IF (NOT(gSystemPrimary.OperatingMode.Stopped)) THEN
	//gMessageManager.register(lCode:=cMCAdviseFunctionalModeNotStationary);
	lDiagnostic := cFunctionalDiagnosticNotStationary;
	request := lDiagnostic;
	RETURN;
END_IF

IF (NOT(lMode.leave())) THEN
	//gMessageManager.register(lCode:=cMCAdviseFunctionalModeWaitingOnPreviousToExit);
	lDiagnostic := cFunctionalDiagnosticWaitingOnPreviousToExit;
	request := lDiagnostic;
	RETURN;
END_IF

lMode REF= mode;
lRequested := TRUE;

IF (NOT(lMode.enter())) THEN
	//gMessageManager.register(lCode:=cMCAdviseFunctionalModeNotYetActive);
	lDiagnostic := cFunctionalDiagnosticNotYetActive;
	request := lDiagnostic;
	RETURN;
END_IF

lDiagnostic := cFunctionalDiagnosticOK;
request := lDiagnostic;


                
END_METHOD

PROPERTY Active : BOOL
GET
                    Active := Mode.Active;
                  
END_GET
END_PROPERTY

(* {attribute 'monitoring' := 'call'} *)
PROPERTY CurrentMode : t_functional_mode
GET
                    CurrentMode := lMode.Mode;


                  
END_GET
SET
                    request(CurrentMode);
                  
END_SET
END_PROPERTY

(* {attribute 'monitoring' := 'call'} *)
PROPERTY Diagnostic : t_functional_diagnostic
GET
                    Diagnostic := lDiagnostic;
                  
END_GET
END_PROPERTY

PROPERTY Mode : REFERENCE TO FunctionalMode
GET
                    Mode REF= lMode;

                  
END_GET
END_PROPERTY

PROPERTY Requested : BOOL
GET
                    Requested := lRequested;
                  
END_GET
END_PROPERTY

PROPERTY TypeToken : t_medium_string
GET
                    TypeToken := 'FuncModeCntrl';
                  
END_GET
END_PROPERTY
END_FUNCTION_BLOCK

FUNCTION_BLOCK FunctionalModeDefault EXTENDS FunctionalMode

            ;
          

METHOD initialize
                  SUPER^.initialize();

lMode := cFunctionalModeDefault;

                
END_METHOD
END_FUNCTION_BLOCK

FUNCTION_BLOCK FunctionalModeLift EXTENDS FunctionalMode

            ;
          

METHOD initialize
                  SUPER^.initialize();

lMode := cFunctionalModeLift;

                
END_METHOD
END_FUNCTION_BLOCK

FUNCTION_BLOCK FunctionalModeTravel EXTENDS FunctionalMode

            ;
          

METHOD initialize
                  SUPER^.initialize();

lMode := cFunctionalModeTravel;

                
END_METHOD
END_FUNCTION_BLOCK

FUNCTION_BLOCK SteerAPositionInterlock EXTENDS WrapperScaledInterlock
  VAR CONSTANT
    cOuterRegion : t_percentage := 1.0;
    cInnerRegion : t_percentage := 0.98;
    cInnerValue : t_percentage := 1.0;
    cOuterValue : t_percentage := 0.0;
    cZeroThreshold : t_percentage := 0.03;
  END_VAR

            ;
          

METHOD initialize
                  Name := 'iSteerAPos';

Input REF= gSystemPrimary.CANOpenMasterDrivePrimary.SteerAngleA.PositionObject;

lTransform.InnerRegion := cInnerRegion;
lTransform.OuterRegion := cOuterRegion;
lTransform.InnerValue := cInnerValue;
lTransform.OuterValue := cOuterValue;

Client.registerServer(gSystemPrimary.Steering.WheelA.Interlock);
Client.ScalingContext REF= gSystemPrimary.Steering.WheelA.InputObject;
Client.ZeroThreshold := cZeroThreshold;
Sign := -1.0;

SUPER^.initialize();

                
END_METHOD
END_FUNCTION_BLOCK

FUNCTION_BLOCK SteerBPositionInterlock EXTENDS WrapperScaledInterlock
  VAR CONSTANT
    cOuterRegion : t_percentage := 1.0;
    cInnerRegion : t_percentage := 0.98;
    cInnerValue : t_percentage := 1.0;
    cOuterValue : t_percentage := 0.0;
    cZeroThreshold : t_percentage := 0.03;
  END_VAR

            ;
          

METHOD initialize
                  Name := 'iSteerBPos';

Input REF= gSystemPrimary.CANOpenMasterDrivePrimary.SteerAngleB.PositionObject;

lTransform.InnerRegion := cInnerRegion;
lTransform.OuterRegion := cOuterRegion;
lTransform.InnerValue := cInnerValue;
lTransform.OuterValue := cOuterValue;

Client.registerServer(gSystemPrimary.Steering.WheelB.Interlock);
Client.ScalingContext REF= gSystemPrimary.Steering.WheelB.InputObject;
Client.ZeroThreshold := cZeroThreshold;
Sign := -1.0;

SUPER^.initialize();

                
END_METHOD
END_FUNCTION_BLOCK

FUNCTION_BLOCK SteerCPositionInterlock EXTENDS WrapperScaledInterlock
  VAR CONSTANT
    cOuterRegion : t_percentage := 1.0;
    cInnerRegion : t_percentage := 0.98;
    cInnerValue : t_percentage := 1.0;
    cOuterValue : t_percentage := 0.0;
    cZeroThreshold : t_percentage := 0.03;
  END_VAR

            ;
          

METHOD initialize
                  Name := 'iSteerCPos';

Input REF= gSystemPrimary.CANOpenMasterDrivePrimary.SteerAngleC.PositionObject;

lTransform.InnerRegion := cInnerRegion;
lTransform.OuterRegion := cOuterRegion;
lTransform.InnerValue := cInnerValue;
lTransform.OuterValue := cOuterValue;

Client.registerServer(gSystemPrimary.Steering.WheelC.Interlock);
Client.ScalingContext REF= gSystemPrimary.Steering.WheelC.InputObject;
Client.ZeroThreshold := cZeroThreshold;
Sign := -1.0;

SUPER^.initialize();

                
END_METHOD
END_FUNCTION_BLOCK

FUNCTION_BLOCK SteerDPositionInterlock EXTENDS WrapperScaledInterlock
  VAR CONSTANT
    cOuterRegion : t_percentage := 1.0;
    cInnerRegion : t_percentage := 0.98;
    cInnerValue : t_percentage := 1.0;
    cOuterValue : t_percentage := 0.0;
    cZeroThreshold : t_percentage := 0.03;
  END_VAR

            ;
          

METHOD initialize
                  Name := 'iSteerDPos';

Input REF= gSystemPrimary.CANOpenMasterDrivePrimary.SteerAngleD.PositionObject;

lTransform.InnerRegion := cInnerRegion;
lTransform.OuterRegion := cOuterRegion;
lTransform.InnerValue := cInnerValue;
lTransform.OuterValue := cOuterValue;

Client.registerServer(gSystemPrimary.Steering.WheelD.Interlock);
Client.ScalingContext REF= gSystemPrimary.Steering.WheelD.InputObject;
Client.ZeroThreshold := cZeroThreshold;
Sign := -1.0;

SUPER^.initialize();

                
END_METHOD
END_FUNCTION_BLOCK

FUNCTION_BLOCK SystemMirrorStandard EXTENDS SystemMirror
  VAR
    lAlarmSubsystem : ReportableAlarmSubsystem;
  END_VAR

            ;
          

METHOD initialize
                  lAlarmSubsystem.initializeState(NopSelf,'',cSCNone);

SUPER^.initialize();
                
END_METHOD

METHOD operator
                  SUPER^.operator();

lSystemState := gSystemPrimary.SystemState.State;
lOperatingMode := gSystemPrimary.OperatingMode.Mode;
lUMFSAllow := gSystemPrimary.lUMFS.Allow;
lGlobalOverride := gManualTemporaryOveride;
lResetDiagnostics := FALSE;
lResetHardware := FALSE;
lResetHealth := FALSE;

(* traffic FROM master PLC *)

(* traffic to master PLC *)

IF (OperatingModeLockRequest) THEN
	gSystemPrimary.OperatingMode.lock(T#2S);
END_IF

IF (OperatingModeRunningRegister) THEN
	gSystemPrimary.OperatingMode.registerRunning();
ELSE
	gSystemPrimary.OperatingMode.registerStopped();
END_IF

IF (UMFSRegister) THEN
	gSystemPrimary.lUMFS.registerSlave();
END_IF

IF (lAlarm<>cSCNone) THEN
	lAlarmSubsystem.SubsystemCode := lAlarm;
	lAlarmSubsystem.report(FALSE);
END_IF

                
END_METHOD
END_FUNCTION_BLOCK

FUNCTION_BLOCK CheckedMovement EXTENDS Movement
  VAR
    lVREnableFunctionalMode : ValueReferenceBool;
    lEnableFunctionalMode : BOOL := TRUE;
    lVREnableUMFSCheck : ValueReferenceBool;
    lEnableUMFSCheck : BOOL := FALSE;
    lChargeInterlock : t_charge_interlock;
    lRegisterPump : BOOL := TRUE;
    lEnableOnlyOnPump : BOOL := TRUE;
    lFunctionalMode : t_functional_mode := cFunctionalModeAny;
    lFunctionalDiagnostic : t_functional_diagnostic := cFunctionalDiagnosticOK;
    lEnableOperatingModeSlow : BOOL := FALSE;
    lEnableUInterfaceSlow : BOOL := FALSE;
    lEnableFunctionSlow : BOOL := FALSE;
    lEnableBeginnerSlow : BOOL := FALSE;
    lUInterfaceSlowFactor : REAL := 1.0;
    lOperatingModeSlowFactor : REAL := 1.0;
    lFunctionSlowFactor : REAL := 1.0;
    lBeginnerSlowFactor : REAL := 1.0;
    lCurrentFunctionSlowFactor : REAL := 1.0;
    lCurrentOperatingModeSlowFactor : REAL := 1.0;
    lCurrentUInterfaceSlowFactor : REAL := 1.0;
    lCurrentBeginnerSlowFactor : REAL := 1.0;
  END_VAR

            ;
          

METHOD checks
                  IF ((lInputResolved<>0) AND (gSystemPrimary.SystemState.State<cSystemStateOperational)) THEN
	Diagnostic := cMovementDiagnosticNotOperational;
	lInputNulled := TRUE;
	//gMessageManager.register(lCode:=cMCAdviseNoFunctionUnlessOperational);
END_IF

IF ((lEnableUMFSCheck) AND (lInputResolved<>0) AND (NOT(gSystemPrimary.lUMFS.Allow))) THEN
	Diagnostic := cMovementDiagnosticUMFS;
	lInputNulled := TRUE;
	//gMessageManager.register(lCode:=cMCAdviseNoFunctionIfUMFS);
END_IF

IF ((lInputResolved<>0) AND (gSystemPrimary.OperatingMode.lMode<cOperatingModeStopped)) THEN
	Diagnostic := cMovementDiagnosticOperatingMode;
	lInputNulled := TRUE;
	//gMessageManager.register(lCode:=cMCAdviseNoFunctionWhenParked);
END_IF

IF (lInputResolved<>0) THEN
	lFunctionalDiagnostic := gSystemPrimary.FunctionalModeControl.request(lFunctionalMode);
	IF ((lFunctionalDiagnostic<>cFunctionalDiagnosticOK) AND
		(lEnableFunctionalMode)) THEN
		Diagnostic := cMovementDiagnosticFunctionalMode;
		lInputNulled := TRUE;
		//gMessageManager.register(lCode:=cMCAdviseNoFunctionWhenParked);
	END_IF
END_IF

IF ((gSystemPrimary.UInterface.IsSlow) AND
	(lEnableUInterfaceSlow)) THEN
	lCurrentUInterfaceSlowFactor := gSystemPrimary.UInterface.SlowFactor * lUInterfaceSlowFactor;
END_IF

IF ((gSystemPrimary.UInterface.IsBeginner) AND
	(lEnableBeginnerSlow)) THEN
	lCurrentBeginnerSlowFactor := lBeginnerSlowFactor;
END_IF

IF ((gSystemPrimary.OperatingMode.IsSlow) AND
	(lEnableOperatingModeSlow)) THEN
	lCurrentOperatingModeSlowFactor := gSystemPrimary.OperatingMode.SlowFactor * lOperatingModeSlowFactor;
END_IF

IF ((lEnableFunctionSlow)) THEN
	lCurrentFunctionSlowFactor := lFunctionSlowFactor;
END_IF

lInputScaling := lInputScaling *
	MIN(MIN(MIN(lCurrentUInterfaceSlowFactor,lCurrentBeginnerSlowFactor),lCurrentOperatingModeSlowFactor),lCurrentFunctionSlowFactor);

lCurrentFunctionSlowFactor := 1.0;
lCurrentOperatingModeSlowFactor := 1.0;
lCurrentUInterfaceSlowFactor := 1.0;

                
END_METHOD

METHOD initialize
                  lVREnableFunctionalMode.initializeValueReference(lEnableFunctionalMode,NopSelf,'EnblFuncMode','Enable functional mode check','',cValueStyleParameter);
lVREnableUMFSCheck.initializeValueReference(lEnableUMFSCheck,NopSelf,'EnblUMFSChk','Enable UMFS check','',cValueStyleParameter);

lChargeInterlock.initializeEventOp(OpSelf,'',cECMovementChargeInterlock);
lChargeInterlock.registerServer(ADR(lInterlock));

SUPER^.initialize();

lRegisterUMFSPrimary := TRUE;
lRegisterUMFSAuxilliary := TRUE;
lRegisterUMFSSecondary := TRUE;

lEnableOperatingModeSlow := TRUE;
lEnableUMFSCheck  := TRUE;

lRegisterActive:= TRUE;
lEnableOnlyOnActiveAllow := TRUE;

lCurrentFunctionSlowFactor := 1.0;
lCurrentOperatingModeSlowFactor := 1.0;
lCurrentUInterfaceSlowFactor := 1.0;

                
END_METHOD

(* {attribute 'monitoring' := 'call'} *)
PROPERTY FunctionalDiagnostic : t_functional_diagnostic
GET
                    FunctionalDiagnostic := lFunctionalDiagnostic;
                  
END_GET
END_PROPERTY

(* {attribute 'monitoring' := 'call'} *)
PROPERTY FunctionalMode : t_functional_mode
GET
                    FunctionalMode := lFunctionalMode;
                  
END_GET
END_PROPERTY

PROPERTY FunctionSlowFactor : REAL
GET
                    FunctionSlowFactor := lFunctionSlowFactor;
                  
END_GET
SET
                    lFunctionSlowFactor := FunctionSlowFactor;
                  
END_SET
END_PROPERTY

PROPERTY OperatingModeSlowFactor : REAL
GET
                    OperatingModeSlowFactor := lOperatingModeSlowFactor;
                  
END_GET
SET
                    lOperatingModeSlowFactor := OperatingModeSlowFactor;
                  
END_SET
END_PROPERTY

PROPERTY TypeToken : t_medium_string
GET
                    TypeToken := 'mChecked';
                  
END_GET
END_PROPERTY

PROPERTY UInterfaceSlowFactor : REAL
GET
                    UInterfaceSlowFactor := lUInterfaceSlowFactor;
                  
END_GET
SET
                    lUInterfaceSlowFactor := UInterfaceSlowFactor;
                  
END_SET
END_PROPERTY

PROPERTY ChargeInterlock : POINTER TO t_charge_interlock
GET
                    ChargeInterlock := ADR(lChargeInterlock);
                  
END_GET
END_PROPERTY
END_FUNCTION_BLOCK

FUNCTION_BLOCK DualMovement EXTENDS CheckedMovement
  VAR
    _Throttle : ThrottleVirtual;
    lMovementA : Movement;
    lScalingA : t_percentage;
    lMovementB : Movement;
    lScalingB : t_percentage;
  END_VAR

            ;
          

METHOD initialize
                  _Throttle.Name := 'Throttle';
lThrottle REF= _Throttle;
registerNonOperational(ADR(_Throttle));

lMovementA.Name := 'mA';
registerNonOperational(ADR(lMovementA));

lMovementA.Name := 'mB';
registerNonOperational(ADR(lMovementB));

SUPER^.initialize();

                
END_METHOD

METHOD operator
                  SUPER^.operator();

lMovementA.InputValue := lThrottle.Value * lScalingA;
lMovementA.operator();

lMovementB.InputValue := lThrottle.Value * lScalingB;
lMovementB.operator();

                
END_METHOD

PROPERTY MovementA : REFERENCE TO Movement
GET
                    MovementA ref= lMovementA;
                  
END_GET
END_PROPERTY

PROPERTY MovementB : REFERENCE TO Movement
GET
                    MovementB ref= lMovementB;
                  
END_GET
END_PROPERTY

(* {attribute 'monitoring' := 'call'} *)
PROPERTY ScalingA : t_percentage
GET
                    ScalingA := lScalingA;
                  
END_GET
SET
                    lScalingA := ScalingA;
                  
END_SET
END_PROPERTY

(* {attribute 'monitoring' := 'call'} *)
PROPERTY ScalingB : t_percentage
GET
                    ScalingB := lScalingB;
                  
END_GET
SET
                    lScalingB := ScalingB;
                  
END_SET
END_PROPERTY

PROPERTY Stalled : BOOL
GET
                    Stalled := ((lMovementA.Stalled) OR
	(lMovementB.Stalled));

                  
END_GET
END_PROPERTY

PROPERTY Stationary : BOOL
GET
                    Stationary := ((lMovementA.Stationary) AND
	(lMovementB.Stationary));

                  
END_GET
END_PROPERTY

PROPERTY TypeToken : t_medium_string
GET
                    TypeToken := 'mDual';
                  
END_GET
END_PROPERTY
END_FUNCTION_BLOCK

FUNCTION_BLOCK Movement EXTENDS OperationalParticleSet
  VAR
    lVREnabledStallManagement : ValueReferenceBool;
    lEnabledStallManagement : BOOL := FALSE;
    lInterlock : t_movement_interlock;
    lInput : ValueObjectPercentageSmoothConditional;
    lInputSecondary : ValueObjectPercentage;
    lEnabled : BOOL := TRUE;
    lForceDisabled : BOOL := FALSE;
    lRegisterUMFSPrimary : BOOL := FALSE;
    lRegisterUMFSAuxilliary : BOOL := FALSE;
    lRegisterUMFSSecondary : BOOL := FALSE;
    lRegisterActive : BOOL := FALSE;
    lEnableOnlyOnActiveAllow : BOOL := FALSE;
    lEnableInputSecondary : BOOL := FALSE;
    lRegisterOperatingMode : BOOL := TRUE;
    lInputScaled : t_percentage;
    lInputResolved : t_percentage;
    lInputProcessed : t_percentage;
    lInputScaling : REAL;
    lInputThresholdAbsolute : t_percentage;
    lVRInputDeadBand : ValueReferencePercentage;
    lInputDeadBand : t_percentage := 0.005;  (* change from 0.05 *)
    lInputScalingOverride : BOOL := FALSE;
    lInputNulled : BOOL;
    lInputPresentAny : BOOL;
    lInputPresentPrimary : BOOL;
    lInputPresentSecondary : BOOL;
    lInputPresentAuxilliary : BOOL;
    lInputPresentAuxilliaryRequest : BOOL;
    lDiagnostic : t_movement_diagnostic;
    _Diagnostic : t_movement_diagnostic;
    lThrottle : REFERENCE TO Throttle;
    lThrottleValue : t_percentage;
    lActive : BOOL;
    lMoving : BOOL;
  END_VAR

            ;
          

METHOD brake
                  
                
END_METHOD

METHOD checks
                  ;
                
END_METHOD

METHOD initialize
                  lVREnabledStallManagement.initializeValueReference(lEnabledStallManagement,NopSelf,'EnblStallMgmt','Enable stall management','',cValueStyleParameter);
lVRInputDeadBand.initializeValueReference(lInputDeadBand,NopSelf,'Deadband','Input deadband','',cValueStyleParameter);

lInterlock.initializeEventOp(OpSelf,'',cECMovementInputInterlock);

lInput.initializeValueObject(NopSelf,'Input','Input value','',cValueStyleConfigurable);
lInputSecondary.initializeValueObject(NopSelf,'InputSecndry','Secondary input value','',cValueStyleConfigurable);

SUPER^.initialize();


                
END_METHOD

METHOD operator
                  lInputNulled := FALSE;
lInputScaling := 1.0;
lInputThresholdAbsolute := 1.0;

lInputResolved := lInput.Value;

IF (ABS(lInput.Value) <= lInputDeadBand) THEN
	lInputPresentPrimary := FALSE;
	
	IF (lInput.Value<>0.0) THEN
		Diagnostic := cMovementDiagnosticDeadband;
		lInputResolved := 0.0;
	END_IF
ELSE
	lInputPresentPrimary := TRUE;
END_IF

IF ((lRegisterUMFSPrimary) AND (lInputPresentPrimary)) THEN
	gSystemPrimary.lUMFS.registerUIPrimary();
END_IF

lInputPresentAuxilliary := lInputPresentAuxilliaryRequest;
lInputPresentAuxilliaryRequest := FALSE;

IF ((lRegisterUMFSAuxilliary) AND (lInputPresentAuxilliary)) THEN
	gSystemPrimary.lUMFS.registerUIAuxilliary();
END_IF

lInputPresentSecondary := FALSE;
IF (lEnableInputSecondary) THEN
	lInputPresentSecondary := (lInputSecondary.Value<>0.0);

	IF (NOT(InputPresentPrimary)) THEN
		lInputResolved := lInputSecondary.Value;
		Diagnostic := cMovementDiagnosticDerived;	
	END_IF

	lEnableInputSecondary := FALSE;
ELSE
	lInputSecondary.Value := 0.0;	
END_IF

IF ((lRegisterUMFSSecondary) AND (lInputPresentSecondary)) THEN
	gSystemPrimary.lUMFS.registerUISecondary();
END_IF

IF (NOT(Enabled)) THEN
	lInputResolved := 0.0;
	lInputPresentPrimary := FALSE;
	lInputPresentSecondary := FALSE;
	lActive := FALSE;
	Diagnostic := cMovementDiagnosticDisabled;
ELSE
	lActive := ((InputPresentPrimary) OR (InputPresentSecondary));
	IF ((lRegisterActive) AND (lActive)) THEN
		gSystemPrimary.Active.registerActive();
	END_IF

	IF (((NOT(gSystemPrimary.Active.Allow)) AND (lEnableOnlyOnActiveAllow))) THEN
		Diagnostic := cMovementDiagnosticActiveDisallow;
		lInputResolved := 0.0;
	END_IF

	checks();

	IF (lInputNulled) THEN
		lInputResolved := 0.0;
	END_IF
END_IF

IF (lInputResolved<>0.0) THEN
	IF (NOT(lInputScalingOverride)) THEN
		lInputProcessed := lInputResolved * lInputScaling;
	ELSE
		lInputProcessed := lInputResolved;
	END_IF
	IF (ABS(lInputProcessed)>lInputThresholdAbsolute) THEN
		lInputProcessed := lInputThresholdAbsolute*lInputProcessed/ABS(lInputProcessed);
		Diagnostic := cMovementDiagnosticThreshold;
	END_IF
ELSE
	lInputProcessed := 0.0;
END_IF

brake();
	
SUPER^.operator();

lThrottleValue := lInterlock.update(lInputProcessed);
IF (lThrottleValue<>lInputProcessed) THEN
	Diagnostic := cMovementDiagnosticInterlock;
END_IF

stall();

lThrottle.Value := lThrottleValue;
lThrottle.operator();

lMoving := FALSE;
IF (lRegisterOperatingMode) THEN
	IF (lThrottle.Value<>0) THEN
		IF (Stalled) THEN
			gSystemPrimary.OperatingMode.registerStalled();
		ELSE
			lMoving := TRUE;
			gSystemPrimary.OperatingMode.registerRunning();
		END_IF
	ELSE
		gSystemPrimary.OperatingMode.registerStopped();
	END_IF
END_IF

lDiagnostic := _Diagnostic;
_Diagnostic := cMovementDiagnosticOK;
lInputScalingOverride := FALSE;
                
END_METHOD

METHOD stall
                  IF ((lEnabledStallManagement) AND 
	(Stalled)) THEN
	lThrottle.Value := 0.0;
	Diagnostic := cMovementDiagnosticStalled;
END_IF
                
END_METHOD

PROPERTY Active : BOOL
GET
                    Active := lActive;
                  
END_GET
END_PROPERTY

PROPERTY CurrentDirection : t_direction
GET
                    CurrentDirection := lThrottle.CurrentDirection;
                  
END_GET
END_PROPERTY

(* {attribute 'monitoring' := 'call'} *)
PROPERTY Diagnostic : t_movement_diagnostic
GET
                    Diagnostic := lDiagnostic;
                  
END_GET
SET
                    _Diagnostic := Diagnostic;
                  
END_SET
END_PROPERTY

PROPERTY Enabled : BOOL
GET
                    Enabled := ((lEnabled) AND (NOT(lForceDisabled)));

                  
END_GET
SET
                    lEnabled := Enabled;
                  
END_SET
END_PROPERTY

PROPERTY EnabledStallManagement : BOOL
GET
                    EnabledStallManagement := lEnabledStallManagement;
                  
END_GET
SET
                    lEnabledStallManagement := EnabledStallManagement;
                  
END_SET
END_PROPERTY

PROPERTY EnableInputSecondary : BOOL
GET
                    EnableInputSecondary := lEnableInputSecondary;
                  
END_GET
SET
                    lEnableInputSecondary := EnableInputSecondary;
                  
END_SET
END_PROPERTY

PROPERTY ForceDisabled : BOOL
GET
                    ForceDisabled := lForceDisabled;
                  
END_GET
SET
                    lForceDisabled := ForceDisabled;

                  
END_SET
END_PROPERTY

(* {attribute 'monitoring' := 'call'} *)
PROPERTY InputDeadBand : t_percentage
GET
                    InputDeadBand := lInputDeadBand;
                  
END_GET
SET
                    lInputDeadBand := abs(InputDeadBand);
                  
END_SET
END_PROPERTY

PROPERTY InputNulled : BOOL
GET
                    InputNulled := lInputNulled;
                  
END_GET
END_PROPERTY

PROPERTY InputObject : REFERENCE TO ValueObjectPercentage
GET
                    InputObject REF= lInput;

                  
END_GET
END_PROPERTY

(* {attribute 'monitoring' := 'call'} *)
PROPERTY InputPresentAny : BOOL
GET
                    InputPresentAny := ((lInputPresentPrimary) OR
	(lInputPresentAuxilliary) OR
	(lInputPresentSecondary));

                  
END_GET
END_PROPERTY

PROPERTY InputPresentAuxilliary : BOOL
GET
                    InputPresentAuxilliary := lInputPresentAuxilliary;

                  
END_GET
END_PROPERTY

PROPERTY InputPresentPrimary : BOOL
GET
                    InputPresentPrimary := lInputPresentPrimary;

                  
END_GET
END_PROPERTY

PROPERTY InputPresentSecondary : BOOL
GET
                    InputPresentSecondary := lInputPresentSecondary;

                  
END_GET
END_PROPERTY

PROPERTY InputProcessed : t_percentage
GET
                    InputProcessed := lInputProcessed;
                  
END_GET
END_PROPERTY

PROPERTY InputResolved : t_percentage
GET
                    InputResolved := lInputResolved;
                  
END_GET
END_PROPERTY

PROPERTY InputScaled : t_percentage
GET
                    InputScaled := lInputScaled;
                  
END_GET
END_PROPERTY

PROPERTY InputScaling : REAL
GET
                    InputScaling := lInputScaling;
                  
END_GET
END_PROPERTY

PROPERTY InputScalingOverride : BOOL
GET
                    InputScalingOverride := lInputScalingOverride;
                  
END_GET
SET
                    lInputScalingOverride := InputScalingOverride;
                  
END_SET
END_PROPERTY

(* {attribute 'monitoring' := 'call'} *)
PROPERTY InputSecondaryValue : t_percentage
GET
                    InputSecondaryValue := lInputSecondary.Value;
                  
END_GET
SET
                    lInputSecondary.Value := InputSecondaryValue;
lInputSecondary.operator();
                  
END_SET
END_PROPERTY

PROPERTY InputThresholdAbsolute : t_percentage
GET
                    InputThresholdAbsolute := lInputThresholdAbsolute;
                  
END_GET
SET
                    lInputThresholdAbsolute := MIN(lInputThresholdAbsolute,ABS(InputThresholdAbsolute));

                  
END_SET
END_PROPERTY

(* {attribute 'monitoring' := 'call'} *)
PROPERTY InputValue : t_percentage
GET
                    InputValue := lInput.Value;
                  
END_GET
SET
                    lInput.Value := InputValue;
                  
END_SET
END_PROPERTY

PROPERTY Interlock : POINTER TO t_movement_interlock
GET
                    Interlock := ADR(lInterlock);
                  
END_GET
END_PROPERTY

PROPERTY Moving : BOOL
GET
                    Moving := lMoving;

                  
END_GET
END_PROPERTY

PROPERTY RequestedDirection : t_direction
GET
                    IF (lInput.Value>0) THEN
	RequestedDirection := cDirectionForward;
ELSIF (lInput.Value<0) THEN
	RequestedDirection := cDirectionReverse;
ELSE
	RequestedDirection := cDirectionStationary;	 
END_IF
                  
END_GET
END_PROPERTY

(* {attribute 'monitoring' := 'call'} *)
PROPERTY Stalled : BOOL
GET
                    IF (__ISVALIDREF(lThrottle)) THEN
	Stalled := lThrottle.Stalled;
ELSE
	Stalled := FALSE;
END_IF
                  
END_GET
END_PROPERTY

(* {attribute 'monitoring' := 'call'} *)
PROPERTY Stationary : BOOL
GET
                    IF (__ISVALIDREF(lThrottle)) THEN
	Stationary := lThrottle.Stationary;
ELSE
	Stationary := FALSE;
END_IF

                  
END_GET
END_PROPERTY

PROPERTY Throttle : REFERENCE TO Throttle
GET
                    Throttle ref= lThrottle;
                  
END_GET
SET
                    lThrottle REF= Throttle;

                  
END_SET
END_PROPERTY

PROPERTY ThrottleValue : t_percentage
GET
                    ThrottleValue := lThrottleValue;
                  
END_GET
END_PROPERTY

PROPERTY TypeToken : t_medium_string
GET
                    TypeToken := 'mMovement';
                  
END_GET
END_PROPERTY
END_FUNCTION_BLOCK

FUNCTION_BLOCK QuadMovement EXTENDS CheckedMovement
  VAR
    _Throttle : ThrottleVirtual;
    lMovementA : Movement;
    lScalingA : t_percentage;
    lMovementB : Movement;
    lScalingB : t_percentage;
    lMovementC : Movement;
    lScalingC : t_percentage;
    lMovementD : Movement;
    lScalingD : t_percentage;
  END_VAR

            ;
          

METHOD initialize
                  _Throttle.Name := 'Throttle';
lThrottle REF= _Throttle;
registerNonOperational(ADR(_Throttle));

lMovementA.Name := 'mA';
registerNonOperational(ADR(lMovementA));

lMovementA.Name := 'mB';
registerNonOperational(ADR(lMovementB));

lMovementA.Name := 'mC';
registerNonOperational(ADR(lMovementC));

lMovementA.Name := 'mD';
registerNonOperational(ADR(lMovementD));

SUPER^.initialize();

                
END_METHOD

METHOD operator
                  SUPER^.operator();

lMovementA.InputValue := lThrottle.Value * lScalingA;
lMovementA.operator();

lMovementB.InputValue := lThrottle.Value * lScalingB;
lMovementB.operator();

lMovementC.InputValue := lThrottle.Value * lScalingC;
lMovementC.operator();

lMovementD.InputValue := lThrottle.Value * lScalingD;
lMovementD.operator();

                
END_METHOD

PROPERTY MovementA : REFERENCE TO Movement
GET
                    MovementA ref= lMovementA;
                  
END_GET
END_PROPERTY

PROPERTY MovementB : REFERENCE TO Movement
GET
                    MovementB ref= lMovementB;
                  
END_GET
END_PROPERTY

PROPERTY MovementC : REFERENCE TO Movement
GET
                    MovementC ref= lMovementC;
                  
END_GET
END_PROPERTY

PROPERTY MovementD : REFERENCE TO Movement
GET
                    MovementD ref= lMovementD;
                  
END_GET
END_PROPERTY

PROPERTY ScalingA : t_percentage
GET
                    ScalingA := lScalingA;
                  
END_GET
SET
                    lScalingA := ScalingA;
                  
END_SET
END_PROPERTY

PROPERTY ScalingB : t_percentage
GET
                    ScalingB := lScalingB;
                  
END_GET
SET
                    lScalingB := ScalingB;
                  
END_SET
END_PROPERTY

PROPERTY ScalingC : t_percentage
GET
                    ScalingC := lScalingC;
                  
END_GET
SET
                    lScalingC := ScalingC;
                  
END_SET
END_PROPERTY

PROPERTY ScalingD : t_percentage
GET
                    ScalingD := lScalingD;
                  
END_GET
SET
                    lScalingD := ScalingD;
                  
END_SET
END_PROPERTY

PROPERTY Stalled : BOOL
GET
                    Stalled := ((lMovementA.Stalled) OR
	(lMovementB.Stalled) OR
	(lMovementC.Stalled) OR
	(lMovementD.Stalled));

                  
END_GET
END_PROPERTY

PROPERTY Stationary : BOOL
GET
                    Stationary := ((lMovementA.Stationary) AND
	(lMovementB.Stationary) AND
	(lMovementC.Stationary) AND
	(lMovementD.Stationary));

                  
END_GET
END_PROPERTY

PROPERTY TypeToken : t_medium_string
GET
                    TypeToken := 'mQuad';
                  
END_GET
END_PROPERTY
END_FUNCTION_BLOCK

FUNCTION_BLOCK AbsoluteThresholdModulation EXTENDS Modulation
  VAR
    lMovement : REFERENCE TO Movement;
    lInitialCutbackThreshold : REAL;
    lCutoutThreshold : REAL;
    lFactor : REAL;
    lOutputThreshold : t_percentage;
  END_VAR

            ;
          

METHOD initialize
                  IF (lCutoutThreshold<=lInitialCutbackThreshold) THEN
	lFactor := 0.0;
ELSE
	lFactor := (-1.0)/(lCutoutThreshold - lInitialCutbackThreshold);
END_IF

                
END_METHOD

METHOD modulate : BOOL
  VAR_INPUT
    input : REAL;
  END_VAR
                  IF ((input>lInitialCutbackThreshold) AND
	(__ISVALIDREF(lMovement)) AND
	(lEnabled)) THEN
	lOutputThreshold := MAX(((input-lInitialCutbackThreshold)*lFactor),0.0);
	
	lMovement.InputThresholdAbsolute := lOutputThreshold;
	modulate := TRUE;	
ELSE
	modulate := FALSE;	
END_IF

                
END_METHOD

PROPERTY CutoutThreshold : REAL
GET
                    CutoutThreshold := lCutoutThreshold;
                  
END_GET
SET
                    lCutoutThreshold := CutoutThreshold;
initialize();
                  
END_SET
END_PROPERTY

PROPERTY Factor : REAL
GET
                    Factor := lFactor;
                  
END_GET
END_PROPERTY

PROPERTY InitialCutbackThreshold : REAL
GET
                    InitialCutbackThreshold := lInitialCutbackThreshold;
                  
END_GET
SET
                    lInitialCutbackThreshold := InitialCutbackThreshold;
initialize();

                  
END_SET
END_PROPERTY

PROPERTY Movement : REFERENCE TO Movement
GET
                    Movement ref= lMovement;
                  
END_GET
SET
                    lMovement REF= Movement;

                  
END_SET
END_PROPERTY

PROPERTY OutputThreshold : t_percentage
GET
                    OutputThreshold := lOutputThreshold;
                  
END_GET
END_PROPERTY
END_FUNCTION_BLOCK

FUNCTION_BLOCK Modulation
  VAR
    lEnabled : BOOL := FALSE;
  END_VAR

            ;
          

METHOD initialize
                  

                
END_METHOD

PROPERTY Enabled : BOOL
GET
                    Enabled := lEnabled;
                  
END_GET
SET
                    lEnabled := Enabled;
                  
END_SET
END_PROPERTY
END_FUNCTION_BLOCK

FUNCTION_BLOCK ProgrammedMovement_LAT0_4WS_Forward EXTENDS ProgrammedMovementTurn

            ;
          

METHOD initialize
                  Name := 'pmtLat04WSFwd';
SUPER^.initialize();

lCode := cProgMovCode_Travel_LAT0_4WS_Forward;

lTargetAngle := 0;
lTargetAngleIncrement := cPi/180.0/3.0;
lTargetAngleZeroThreshold := 0.005;
lTravelThrottle := 0.05;
	
lSteerModeRequired := cSteerModeLateral;
lSteerModeOnFinishing := cSteerMode4WS;

                
END_METHOD
END_FUNCTION_BLOCK

FUNCTION_BLOCK ProgrammedMovement_LAT0_4WS_Reverse EXTENDS ProgrammedMovementTurn

            ;
          

METHOD initialize
                  Name := 'pmtLat04WSRev';
SUPER^.initialize();

lCode := cProgMovCode_Travel_LAT0_4WS_Reverse;

lTargetAngle := 0;
lTargetAngleIncrement := cPi/180.0/3.0;
lTargetAngleZeroThreshold := 0.005;
lTravelThrottle := -0.05;
	
lSteerModeRequired := cSteerModeLateral;
lSteerModeOnFinishing := cSteerMode4WS;

                
END_METHOD
END_FUNCTION_BLOCK

FUNCTION_BLOCK ProgrammedMovement_LAT0_Forward EXTENDS ProgrammedMovementTurn

            ;
          

METHOD initialize
                  Name := 'pmtLat0Fwd';
SUPER^.initialize();

lCode := cProgMovCode_Travel_LAT0_Forward;

lTargetAngle := 0;
lTargetAngleIncrement := cPi/180.0/3.0;
lTargetAngleZeroThreshold := 0.005;
lTravelThrottle := 0.05;
	
lSteerModeRequired := cSteerModeLateral;
lSteerModeOnFinishing := cSteerModeLateral;
                
END_METHOD
END_FUNCTION_BLOCK

FUNCTION_BLOCK ProgrammedMovement_LAT0_Reverse EXTENDS ProgrammedMovementTurn

            ;
          

METHOD initialize
                  Name := 'pmtLat0Rev';
SUPER^.initialize();

lCode := cProgMovCode_Travel_LAT0_Reverse;

lTargetAngle := 0;
lTargetAngleIncrement := cPi/180.0/3.0;
lTargetAngleZeroThreshold := 0.005;
lTravelThrottle := -0.05;
	
lSteerModeRequired := cSteerModeLateral;
lSteerModeOnFinishing := cSteerModeLateral;
                
END_METHOD
END_FUNCTION_BLOCK

FUNCTION_BLOCK ProgrammedMovement_LATNeg90_Forward EXTENDS ProgrammedMovementTurn

            ;
          

METHOD initialize
                  Name := 'pmtLat-90Fwd';
SUPER^.initialize();

lCode := cProgMovCode_Travel_LATNeg90_Forward;

lTargetAngle := -1.0*cPiOn2*85.0/90.0;
lTargetAngleIncrement := cPi/180.0/3.0;
lTargetAngleZeroThreshold := 0.005;
lTravelThrottle := 0.05;
	
lSteerModeRequired := cSteerModeLateral;
lSteerModeOnFinishing := cSteerModeLateral;
                
END_METHOD
END_FUNCTION_BLOCK

FUNCTION_BLOCK ProgrammedMovement_LATNeg90_Reverse EXTENDS ProgrammedMovementTurn

            ;
          

METHOD initialize
                  Name := 'pmtLat-90Rev';
SUPER^.initialize();

lCode := cProgMovCode_Travel_LATNeg90_Reverse;

lTargetAngle := -1.0*cPiOn2*85.0/90.0;
lTargetAngleIncrement := cPi/180.0/3.0;
lTargetAngleZeroThreshold := 0.005;
lTravelThrottle := -0.05;
	
lSteerModeRequired := cSteerModeLateral;
lSteerModeOnFinishing := cSteerModeLateral;
                
END_METHOD
END_FUNCTION_BLOCK

FUNCTION_BLOCK ProgrammedMovement_LATPos90_Forward EXTENDS ProgrammedMovementTurn

            ;
          

METHOD initialize
                  Name := 'pmtLat90Fwd';
SUPER^.initialize();

lCode := cProgMovCode_Travel_LATPos90_Forward;

lTargetAngle := cPiOn2*85.0/90.0;
lTargetAngleIncrement := cPi/180.0/3.0;
lTargetAngleZeroThreshold := 0.005;
lTravelThrottle := 0.05;
	
lSteerModeRequired := cSteerModeLateral;
lSteerModeOnFinishing := cSteerModeLateral;
                
END_METHOD
END_FUNCTION_BLOCK

FUNCTION_BLOCK ProgrammedMovement_LATPos90_Reverse EXTENDS ProgrammedMovementTurn

            ;
          

METHOD initialize
                  Name := 'pmtLat90Rev';
SUPER^.initialize();

lCode := cProgMovCode_Travel_LATPos90_Reverse;

lTargetAngle := cPiOn2*85.0/90.0;
lTargetAngleIncrement := cPi/180.0/3.0;
lTargetAngleZeroThreshold := 0.005;
lTravelThrottle := -0.05;
	
lSteerModeRequired := cSteerModeLateral;
lSteerModeOnFinishing := cSteerModeLateral;
                
END_METHOD
END_FUNCTION_BLOCK

FUNCTION_BLOCK ProgrammedMovement_Steer_0 EXTENDS ProgrammedMovementSteer

            ;
          

METHOD initialize
                  Name := 'pms0';
SUPER^.initialize();

lCode := cProgMovCode_Steer_0;

lTargetAngle := 0;
lTargetAngleIncrement := cPi/180.0/3.0;
lTargetAngleZeroThreshold := 0.005;

                
END_METHOD
END_FUNCTION_BLOCK

FUNCTION_BLOCK ProgrammedMovement_Test1 EXTENDS ProgrammedMovementMulti

            ;
          

METHOD initialize
                  Name := 'ProgMovTest1';

SUPER^.initialize();
SubSystem := cSubsystemTravel;

lCode := cProgMovCode_Test1;
lTimeStepMax := 2000;

registerMovement(cProgMovCode_Travel_LATPos90_Forward);
registerMovement(cProgMovCode_Travel_LAT0_Forward);
                
END_METHOD
END_FUNCTION_BLOCK

FUNCTION_BLOCK ProgrammedMovement EXTENDS CheckedMovement
  VAR CONSTANT
    cInactiveTimer : t_time := TIME#2m0s0ms;
  END_VAR
  VAR
    _Throttle : ThrottleVirtual;
    lCode : t_prog_mov_code;
    lState : t_prog_mov_state;
    lSuccess : BOOL := FALSE;
    lProgMovDiagnostic : t_prog_mov_diagnostic;
    _ProgMovDiagnostic : t_prog_mov_diagnostic;
    lTimeStep : UINT;
    lTimeStepMax : UINT := 1000;
    lInactiveTimer : t_timer;
  END_VAR

            ;
          

METHOD disabled
                  lInactiveTimer.reset();
lSuccess := FALSE;
lTimeStep := 0;
	
IF (Enabled) THEN
	ProgMovDiagnostic := cProgMovDiagnosticEnabling;
	lState := cProgMovStatePreparing;
END_IF
                
END_METHOD

METHOD finishing
                  IF (LeavingCondition) THEN
	ProgMovDiagnostic := cProgMovDiagnosticLeaving;
	lState := cProgMovStateLeaving;
END_IF

IF (InterruptCondition) THEN
	ProgMovDiagnostic := cProgMovDiagnosticInterrupted;
	lState := cProgMovStateLeaving;
END_IF

                
END_METHOD

METHOD inactive
                  IF (ActiveCondition) THEN
	ProgMovDiagnostic := cProgMovDiagnosticActivating;
	lState := cProgMovStateWaiting;
END_IF

lInactiveTimer.operator();
IF (lInactiveTimer.Expired) THEN
	lEnabled := FALSE;
	lState := cProgMovStateDisabled;
	ProgMovDiagnostic := cProgMovDiagnosticInactiveTimeout;
END_IF
                
END_METHOD

METHOD initialize
                  Name := 'ProgMov';

_Throttle.Name := 'Throttle';
lThrottle REF= _Throttle;
registerNonOperational(ADR(_Throttle));

SUPER^.initialize();

lEnabledStallManagement := FALSE;
lRegisterOperatingMode := FALSE;
lEnableOnlyOnActiveAllow := FALSE;

lInactiveTimer.initialize();
lInactiveTimer.Enable := TRUE;
lInactiveTimer.Period := cInactiveTimer;


                
END_METHOD

METHOD leaving
                  IF (LeavingCompleteCondition) THEN
	lEnabled := FALSE;
	lState := cProgMovStateDisabled;
	ProgMovDiagnostic := cProgMovDiagnosticLeaving;
END_IF
                
END_METHOD

METHOD operator
                  SUPER^.operator();

IF (NOT(Enabled)) THEN
	lState := cProgMovStateDisabled;
END_IF

CASE (lState) OF
	cProgMovStateDisabled:
		disabled();

	cProgMovStatePreparing:
		preparing();
	
	cProgMovStateInactive:
		inactive();
	
	cProgMovStateWaiting:
		waiting();
	
	cProgMovStateRunning:
		running();
	
	cProgMovStateFinishing:
		finishing();
		
	cProgMovStateLeaving:
		leaving();	
END_CASE

lProgMovDiagnostic := _ProgMovDiagnostic;
_ProgMovDiagnostic := cProgMovDiagnosticDisabled;

                
END_METHOD

METHOD preparing
                  IF (PreparedCondition) THEN
	ProgMovDiagnostic := cProgMovDiagnosticPrepared;
	lState := cProgMovStateInactive;
END_IF

                
END_METHOD

METHOD running
                  ProgMovDiagnostic := cProgMovDiagnosticRunning;
lTimeStep := lTimeStep + 1;

IF (NOT(ActiveCondition)) THEN
	ProgMovDiagnostic := cProgMovDiagnosticDeactivatingFromRunning;
	lState := cProgMovStateFinishing;
END_IF

IF (InterruptCondition) THEN
	ProgMovDiagnostic := cProgMovDiagnosticInterrupted;
	lState := cProgMovStateLeaving;
END_IF

IF (FinishCondition) THEN
	ProgMovDiagnostic := cProgMovDiagnosticFinishing;
	lState := cProgMovStateFinishing;
	lSuccess := TRUE;
END_IF


                
END_METHOD

METHOD waiting
                  IF (NOT(ActiveCondition)) THEN
	ProgMovDiagnostic := cProgMovDiagnosticDeactivatingFromWaiting;
	lState := cProgMovStateInactive;
END_IF

IF (StartCondition) THEN
	ProgMovDiagnostic := cProgMovDiagnosticStarting;
	lState := cProgMovStateRunning;
	
	lSuccess := FALSE;
	lTimeStep := 0;
END_IF
                
END_METHOD

(* {attribute 'monitoring' := 'call'} *)
PROPERTY ActiveCondition : BOOL
GET
                    ActiveCondition := true;
                  
END_GET
END_PROPERTY

(* {attribute 'monitoring' := 'call'} *)
PROPERTY Available : BOOL
GET
                    Available := NOT(ForceDisabled);
                  
END_GET
END_PROPERTY

PROPERTY Code : t_prog_mov_code
GET
                    Code := lCode;
                  
END_GET
SET
                    lCode := Code;
                  
END_SET
END_PROPERTY

(* {attribute 'monitoring' := 'call'} *)
PROPERTY FinishCondition : BOOL
GET
                    FinishCondition := (lTimeStep>lTimeStepMax);

                  
END_GET
END_PROPERTY

(* {attribute 'monitoring' := 'call'} *)
PROPERTY InterruptCondition : BOOL
GET
                    InterruptCondition := FALSE;

IF (gSystemPrimary.UInterface.JoystickInputPresent) THEN
	InterruptCondition := TRUE;	
END_IF
                  
END_GET
END_PROPERTY

(* {attribute 'monitoring' := 'call'} *)
PROPERTY LeavingCompleteCondition : BOOL
GET
                    LeavingCompleteCondition := true;
                  
END_GET
END_PROPERTY

(* {attribute 'monitoring' := 'call'} *)
PROPERTY LeavingCondition : BOOL
GET
                    LeavingCondition := true;
                  
END_GET
END_PROPERTY

(* {attribute 'monitoring' := 'call'} *)
PROPERTY PreparedCondition : BOOL
GET
                    PreparedCondition := TRUE;
                  
END_GET
END_PROPERTY

(* {attribute 'monitoring' := 'call'} *)
PROPERTY ProgMovDiagnostic : t_prog_mov_diagnostic
GET
                    ProgMovDiagnostic := lProgMovDiagnostic;
                  
END_GET
SET
                    _ProgMovDiagnostic := ProgMovDiagnostic;
                  
END_SET
END_PROPERTY

(* {attribute 'monitoring' := 'call'} *)
PROPERTY StartCondition : BOOL
GET
                    StartCondition := FALSE;

                  
END_GET
END_PROPERTY

PROPERTY State : t_prog_mov_state
GET
                    State := lState;
                  
END_GET
END_PROPERTY

PROPERTY TimeStepMax : UINT
GET
                    TimeStepMax := lTimeStepMax;
                  
END_GET
SET
                    lTimeStepMax := TimeStepMax;
                  
END_SET
END_PROPERTY

PROPERTY TypeToken : t_medium_string
GET
                    TypeToken := 'mProgrammed';
                  
END_GET
END_PROPERTY
END_FUNCTION_BLOCK

FUNCTION_BLOCK ProgrammedMovementControl EXTENDS NonOperationalParticleSet
  VAR
    lProgMovNull : ProgrammedMovementNull;
    lProgMov_Steer_0 : ProgrammedMovementSteer;
    lMovement : REFERENCE TO ProgrammedMovement;  (* lProgMov_Test1: ProgrammedMovementMulti; *)
    lDiagnostic : t_functional_diagnostic;
    lRequested : BOOL := FALSE;
  END_VAR

            ;
          

METHOD getMovement : REFERENCE TO ProgrammedMovement
  VAR_INPUT
    code : t_prog_mov_code;
  END_VAR
                  getMovement REF= lProgMovNull;

CASE code OF		
		
	(*
cProgMovCode_Lift_Top:
		getMovement REF= lProgMov_Lift_Top;	

	cProgMovCode_Lift_Bottom:
		getMovement REF= lProgMov_Lift_Bottom;	
	
	cProgMovCode_Lift_StandardOnGround:
		getMovement REF= lProgMov_Lift_StandardOnGround;	
		
	cProgMovCode_Lift_StandardGround:
		getMovement REF= lProgMov_Lift_StandardGround;	
		
	cProgMovCode_Lift_StandardTruck:
		getMovement REF= lProgMov_Lift_StandardTruck;	

	cProgMovCode_Lift_StandardStack1:
		getMovement REF= lProgMov_Lift_StandardStack1;	
		
	cProgMovCode_Lift_StandardStack2:
		getMovement REF= lProgMov_Lift_StandardStack2;	

	cProgMovCode_Lift_HicubeOnGround:
		getMovement REF= lProgMov_Lift_HicubeOnGround;	
		
	cProgMovCode_Lift_HicubeGround:
		getMovement REF= lProgMov_Lift_HicubeGround;	
		
	cProgMovCode_Lift_HicubeTruck:
		getMovement REF= lProgMov_Lift_HicubeTruck;	

	cProgMovCode_Lift_HicubeStack1:
		getMovement REF= lProgMov_Lift_HicubeStack1;	

	cProgMovCode_Lift_HicubeStack2:
		getMovement REF= lProgMov_Lift_HicubeStack2;	
				
	cProgMovCode_Travel_LAT0_Forward:
		getMovement REF= lProgMov_Travel_LAT0_Forward;		

	cProgMovCode_Travel_LAT0_Reverse:
		getMovement REF= lProgMov_Travel_LAT0_Reverse;		

	cProgMovCode_Travel_LAT0_4WS_Forward:
		getMovement REF= lProgMov_Travel_LAT0_4WS_Forward;		

	cProgMovCode_Travel_LAT0_4WS_Reverse:
		getMovement REF= lProgMov_Travel_LAT0_4WS_Reverse;		

	cProgMovCode_Travel_LATPos90_Forward:
		getMovement REF= lProgMov_Travel_LATPos90_Forward;

	cProgMovCode_Travel_LATPos90_Reverse:
		getMovement REF= lProgMov_Travel_LATPos90_Reverse;

	cProgMovCode_Travel_LATNeg90_Forward:
		getMovement REF= lProgMov_Travel_LATNeg90_Forward;

	cProgMovCode_Travel_LATNeg90_Reverse:
		getMovement REF= lProgMov_Travel_LATNeg90_Reverse;

	cProgMovCode_Test1:
		getMovement REF= lProgMov_Test1;*)

	cProgMovCode_Steer_0:
		getMovement REF= lProgMov_Steer_0;
END_CASE

                
END_METHOD

METHOD initialize
                  Name := 'ProgMovCntrl';

registerNonOperational(ADR(lProgMovNull));

lProgMov_Steer_0.Code := cProgMovCode_Steer_0;
lProgMov_Steer_0.Name := gTypeHandler.getTokenForEnum(cEnumTypeProgMovCode,cProgMovCode_Steer_0);
lProgMov_Steer_0.TargetAngle := 0;
lProgMov_Steer_0.TargetAngleIncrement := cPi/180.0/3.0;
lProgMov_Steer_0.TargetAngleZeroThreshold := 0.005;
registerNonOperational(ADR(lProgMov_Steer_0));

(*lProgMov_Test1.Code := cProgMovCode_Test1;
lProgMov_Test1.Name := getStringForProgMovCode(cProgMovCode_Test1);
lProgMov_Test1.TimeStepMax := 2000;
lProgMov_Test1.registerMovement(cProgMovCode_Travel_LATPos90_Forward);
lProgMov_Test1.registerMovement(cProgMovCode_Travel_LAT0_Forward);
registerNonOperational(ADR(lProgMov_Test1));*)

lMovement REF= lProgMovNull;

SUPER^.initialize();
SubSystem := cSubsystemMachine;


                
END_METHOD

METHOD operator
                  request(gSystemPrimary.UInterface.AutomationRequest);

IF ((NOT(lMovement.Enabled)) OR
	(gSystemPrimary.SystemState.State<cSystemStateOperational)) THEN
	lMovement REF= lProgMovNull;
END_IF

lMovement.operator();
                
END_METHOD

METHOD request
  VAR_INPUT
    requested : t_prog_mov_code;
  END_VAR
  VAR
    movement : REFERENCE TO ProgrammedMovement;
  END_VAR
                  IF (requested=cProgMovCodeNone) THEN
	RETURN;
END_IF

IF (requested=cProgMovCode_Clear) THEN
	lMovement REF= lProgMovNull;
	RETURN;
END_IF

movement REF= getMovement(requested);
IF (NOT(__ISVALIDREF(movement))) THEN
	RETURN;
END_IF

IF (movement.Code=cProgMovCodeNone) THEN
	RETURN;
END_IF

IF (NOT(movement.Available)) THEN
	RETURN;
END_IF

movement.Enabled := TRUE;
IF (NOT(movement.Enabled)) THEN
	movement.Enabled := FALSE;
	RETURN;
END_IF

lMovement REF= movement;

// allows continuous request, will not abort if requesting current

                
END_METHOD

(* {attribute 'monitoring' := 'call'} *)
PROPERTY CurrentMovement : t_prog_mov_code
GET
                    CurrentMovement := lMovement.Code;


                  
END_GET
SET
                    request(CurrentMovement);
                  
END_SET
END_PROPERTY

PROPERTY CurrentState : t_prog_mov_state
GET
                    CurrentState := lMovement.State;
                  
END_GET
END_PROPERTY

PROPERTY Enabled : BOOL
GET
                    Enabled := (lMovement.Enabled);
                  
END_GET
END_PROPERTY

PROPERTY Movement : REFERENCE TO ProgrammedMovement
GET
                    Movement REF= lMovement;

                  
END_GET
END_PROPERTY

PROPERTY Requested : BOOL
GET
                    Requested := lRequested;
                  
END_GET
END_PROPERTY

PROPERTY TypeToken : t_medium_string
GET
                    TypeToken := 'mProgCntrl';
                  
END_GET
END_PROPERTY
END_FUNCTION_BLOCK

FUNCTION_BLOCK ProgrammedMovementMulti EXTENDS ProgrammedMovement
  VAR CONSTANT
    cCOuntMax : USINT := 32;
  END_VAR
  VAR
    lProgMovNull : ProgrammedMovementNull;
    lMovement : REFERENCE TO ProgrammedMovement;
    lSequence : t_pmc_set;
    lCount : USINT := 0;
    lCurrent : USINT := 0;
    lSequenceAchieved : BOOL := FALSE;
  END_VAR

            ;
          

METHOD disabled
                  SUPER^.disabled();

lSequenceAchieved := FALSE;
lMovement REF= lProgMovNull;

                
END_METHOD

METHOD initialize
                  Name := 'ProgMovMulti';

registerNonOperational(ADR(lProgMovNull));

lMovement REF= lProgMovNull;

SUPER^.initialize();



                
END_METHOD

METHOD next
                  IF (lCurrent>=lCount) THEN
	lSequenceAchieved := TRUE;
	lMovement REF= lProgMovNull;
	RETURN;
END_IF

lCurrent := lCurrent + 1;
request(lSequence[lCurrent]);

                
END_METHOD

METHOD registerMovement
  VAR_INPUT
    code : t_prog_mov_code;
  END_VAR
                  IF (lCount>=cCOuntMax) THEN
	gCodeErrorHandler(pMessage:=CONCAT('exceeded sequence size in ',lIdentity));
	RETURN;
END_IF

lCount := lCount+1;
lSequence[lCount] := code;
                
END_METHOD

METHOD request
  VAR_INPUT
    code : t_prog_mov_code;
  END_VAR
  VAR
    movement : REFERENCE TO ProgrammedMovement;
  END_VAR
                  lMovement REF= lProgMovNull;

movement REF= gSystemPrimary.ProgrammedMovementControl.getMovement(code);
	
IF (NOT(__ISVALIDREF(movement))) THEN
	lSequenceAchieved := TRUE;
	RETURN;
END_IF

IF (movement.Code=cProgMovCodeNone) THEN
	lSequenceAchieved := TRUE;
	RETURN;
END_IF

IF (NOT(movement.Available)) THEN
	lSequenceAchieved := TRUE;
	RETURN;
END_IF

movement.Enabled := TRUE;
IF (NOT(movement.Enabled)) THEN
	movement.Enabled := FALSE;
	lSequenceAchieved := TRUE;
	RETURN;
END_IF

lMovement REF= movement;

                
END_METHOD

METHOD running
                  SUPER^.running();

IF (lState<>cProgMovStateRunning) THEN
	RETURN;
END_IF

IF (not(lMovement.Enabled)) THEN
	next();
	RETURN;
END_IF

lMovement.operator();

                
END_METHOD

METHOD waiting
                  IF (NOT(ActiveCondition)) THEN
	ProgMovDiagnostic := cProgMovDiagnosticDeactivatingFromWaiting;
	lState := cProgMovStateInactive;
END_IF

IF (StartCondition) THEN
	ProgMovDiagnostic := cProgMovDiagnosticStarting;
	lState := cProgMovStateRunning;
	
	lSuccess := FALSE;
	lTimeStep := 0;
END_IF

lCurrent := 0;
                
END_METHOD

(* {attribute 'monitoring' := 'call'} *)
PROPERTY FinishCondition : BOOL
GET
                    FinishCondition := ((lSequenceAchieved) OR
	(lTimeStep>lTimeStepMax));

                  
END_GET
END_PROPERTY

(* {attribute 'monitoring' := 'call'} *)
PROPERTY InterruptCondition : BOOL
GET
                    InterruptCondition := FALSE;

IF ((gSystemPrimary.UInterface.TravelJoystickInputPresent) AND
	(gSystemPrimary.UInterface.LiftJoystickInputPresent)) THEN
	InterruptCondition := TRUE;	
END_IF
                  
END_GET
END_PROPERTY

(* {attribute 'monitoring' := 'call'} *)
PROPERTY StartCondition : BOOL
GET
                    StartCondition := gSystemPrimary.UInterface.AutomationStart;

                  
END_GET
END_PROPERTY

PROPERTY TypeToken : t_medium_string
GET
                    TypeToken := 'mProgMulti';
                  
END_GET
END_PROPERTY
END_FUNCTION_BLOCK

FUNCTION_BLOCK ProgrammedMovementNull EXTENDS ProgrammedMovement

            ;
          

METHOD initialize
                  Name := 'ProgMovNull';

SUPER^.initialize();
SubSystem := cSubsystemMachine;

lCode := cProgMovCodeNone;

lSuccess := FALSE;
lEnabled := FALSE;
lState := cProgMovStateDisabled;
lProgMovDiagnostic := cProgMovDiagnosticDisabled;

                
END_METHOD

METHOD operator
                  lEnabled := FALSE;

                
END_METHOD
END_FUNCTION_BLOCK

FUNCTION_BLOCK ProgrammedMovementSteer EXTENDS ProgrammedMovement
  VAR
    lTargetAngle : REAL := 0;
    lTargetAngleIncrement : REAL := 0;
    lTargetAngleZeroThreshold : REAL := 0.001;
    lTargetAngleAchieved : BOOL;
  END_VAR

            ;
          

METHOD disabled
                  SUPER^.disabled();

lTargetAngleAchieved := FALSE;

                
END_METHOD

METHOD finishing
                  SUPER^.finishing();

IF (lState<>cProgMovStateFinishing) THEN
	RETURN;
END_IF


                
END_METHOD

METHOD initialize
                  Name := 'ProgMovSteer';

SUPER^.initialize();
SubSystem := cSubsystemSteer;

                
END_METHOD

METHOD operator
                  // lInput.Value := BOOL_TO_REAL(gSystemPrimary.UInterface.AutomationStart);

SUPER^.operator();

                
END_METHOD

METHOD running
                  SUPER^.running();

IF (lState<>cProgMovStateRunning) THEN
	RETURN;
END_IF

IF (ABS(gSystemPrimary.Steering.TargetAngle-lTargetAngle)<=lTargetAngleZeroThreshold) THEN
	lTargetAngleAchieved := TRUE;
ELSE
	lTargetAngleAchieved := FALSE;

	IF (gSystemPrimary.Steering.TargetAngle < lTargetAngle) THEN
		gSystemPrimary.Steering.TargetAngleIncrementDerived := lTargetAngleIncrement;
		gSystemPrimary.Steering.EnableDerivedTargetAngleIncrement := TRUE;
	END_IF
	IF (gSystemPrimary.Steering.TargetAngle > lTargetAngle) THEN
		gSystemPrimary.Steering.TargetAngleIncrementDerived := 0.0 - lTargetAngleIncrement;
		gSystemPrimary.Steering.EnableDerivedTargetAngleIncrement := TRUE;
	END_IF
END_IF

                
END_METHOD

METHOD waiting
                  IF (NOT(ActiveCondition)) THEN
	ProgMovDiagnostic := cProgMovDiagnosticDeactivatingFromWaiting;
	lState := cProgMovStateInactive;
END_IF

IF (StartCondition) THEN
	ProgMovDiagnostic := cProgMovDiagnosticStarting;
	lState := cProgMovStateRunning;
	
	lSuccess := FALSE;
	lTimeStep := 0;
END_IF

                
END_METHOD

(* {attribute 'monitoring' := 'call'} *)
PROPERTY FinishCondition : BOOL
GET
                    FinishCondition := ((lTargetAngleAchieved) OR
	(lTimeStep>lTimeStepMax));

                  
END_GET
END_PROPERTY

(* {attribute 'monitoring' := 'call'} *)
PROPERTY InterruptCondition : BOOL
GET
                    InterruptCondition := FALSE;

IF (gSystemPrimary.Steering.InputPresentPrimary) THEN
	InterruptCondition := TRUE;	
END_IF
                  
END_GET
END_PROPERTY

(* {attribute 'monitoring' := 'call'} *)
PROPERTY LeavingCondition : BOOL
GET
                    LeavingCondition := true;
                  
END_GET
END_PROPERTY

(* {attribute 'monitoring' := 'call'} *)
PROPERTY StartCondition : BOOL
GET
                    StartCondition := TRUE;

                  
END_GET
END_PROPERTY

PROPERTY TargetAngle : REAL
GET
                    TargetAngle := lTargetAngle;
                  
END_GET
SET
                    lTargetAngle := TargetAngle;
                  
END_SET
END_PROPERTY

PROPERTY TargetAngleIncrement : REAL
GET
                    TargetAngleIncrement := lTargetAngleIncrement;
                  
END_GET
SET
                    lTargetAngleIncrement := TargetAngleIncrement;
                  
END_SET
END_PROPERTY

PROPERTY TargetAngleZeroThreshold : REAL
GET
                    TargetAngleZeroThreshold := lTargetAngleZeroThreshold;
                  
END_GET
SET
                    lTargetAngleZeroThreshold := TargetAngleZeroThreshold;
                  
END_SET
END_PROPERTY

PROPERTY TypeToken : t_medium_string
GET
                    TypeToken := 'mProgSteer';
                  
END_GET
END_PROPERTY
END_FUNCTION_BLOCK

FUNCTION_BLOCK ProgrammedMovementTurn EXTENDS ProgrammedMovement
  VAR
    lTargetAngle : REAL := 0;
    lTargetAngleIncrement : REAL := 0;
    lTargetAngleZeroThreshold : REAL := 0.001;
    lTravelThrottle : t_percentage := 0.0;
    lSteerModeRequired : t_steer_mode := cSteerModeNone;
    lSteerModeOnFinishing : t_steer_mode := cSteerModeNone;
    lTargetAngleAchieved : BOOL;
  END_VAR

            ;
          

METHOD disabled
                  SUPER^.disabled();

lTargetAngleAchieved := FALSE;

                
END_METHOD

METHOD finishing
                  SUPER^.finishing();

IF (lState<>cProgMovStateFinishing) THEN
	RETURN;
END_IF

IF (gSystemPrimary.Steering.CurrentMode<>lSteerModeOnFinishing) THEN
	gSystemPrimary.Steering.requestSteerMode(lSteerModeOnFinishing);
END_IF

                
END_METHOD

METHOD initialize
                  Name := 'ProgMovTurn';

SUPER^.initialize();
SubSystem := cSubsystemTravel;

                
END_METHOD

METHOD operator
                  lInput.Value := BOOL_TO_REAL(gSystemPrimary.UInterface.AutomationStart);

SUPER^.operator();

                
END_METHOD

METHOD running
                  SUPER^.running();

IF (lState<>cProgMovStateRunning) THEN
	RETURN;
END_IF

IF (ABS(gSystemPrimary.Steering.TargetAngle-lTargetAngle)<=lTargetAngleZeroThreshold) THEN
	lTargetAngleAchieved := TRUE;
ELSE
	lTargetAngleAchieved := FALSE;

	IF (gSystemPrimary.Steering.TargetAngle < lTargetAngle) THEN
		gSystemPrimary.Steering.TargetAngleIncrementDerived := lTargetAngleIncrement;
		gSystemPrimary.Steering.EnableDerivedTargetAngleIncrement := TRUE;
	END_IF
	IF (gSystemPrimary.Steering.TargetAngle > lTargetAngle) THEN
		gSystemPrimary.Steering.TargetAngleIncrementDerived := 0.0 - lTargetAngleIncrement;
		gSystemPrimary.Steering.EnableDerivedTargetAngleIncrement := TRUE;
	END_IF
END_IF

gSystemPrimary.Travel.EnableInputSecondary := TRUE;
gSystemPrimary.Travel.InputScalingOverride := TRUE;
gSystemPrimary.Travel.InputSecondaryValue := lTravelThrottle;
                
END_METHOD

METHOD waiting
                  IF (NOT(ActiveCondition)) THEN
	ProgMovDiagnostic := cProgMovDiagnosticDeactivatingFromWaiting;
	lState := cProgMovStateInactive;
END_IF

IF (StartCondition) THEN
	ProgMovDiagnostic := cProgMovDiagnosticStarting;
	lState := cProgMovStateRunning;
	
	lSuccess := FALSE;
	lTimeStep := 0;
END_IF

IF (gSystemPrimary.Steering.CurrentMode<>lSteerModeRequired) THEN
	gSystemPrimary.Steering.requestSteerMode(lSteerModeRequired);
END_IF
                
END_METHOD

(* {attribute 'monitoring' := 'call'} *)
PROPERTY FinishCondition : BOOL
GET
                    FinishCondition := (((lTargetAngleAchieved) AND
	(gSystemPrimary.Steering.OK)) OR
	(lTimeStep>lTimeStepMax));

                  
END_GET
END_PROPERTY

(* {attribute 'monitoring' := 'call'} *)
PROPERTY InterruptCondition : BOOL
GET
                    InterruptCondition := FALSE;

IF (gSystemPrimary.UInterface.TravelJoystickInputPresent) THEN
	InterruptCondition := TRUE;	
END_IF
                  
END_GET
END_PROPERTY

(* {attribute 'monitoring' := 'call'} *)
PROPERTY LeavingCondition : BOOL
GET
                    LeavingCondition := ((gSystemPrimary.Steering.CurrentMode=lSteerModeOnFinishing) AND
	(gSystemPrimary.Steering.OK));
                  
END_GET
END_PROPERTY

(* {attribute 'monitoring' := 'call'} *)
PROPERTY StartCondition : BOOL
GET
                    StartCondition := ((gSystemPrimary.Steering.CurrentMode=lSteerModeRequired) AND
	(gSystemPrimary.Steering.OK) AND
	(gSystemPrimary.UInterface.AutomationStart) AND
	((gSystemPrimary.Travel.CurrentDirection=cDirectionStationary) OR
	((gSystemPrimary.Travel.CurrentDirection=cDirectionForward) AND (lTravelThrottle>0.0)) OR
	((gSystemPrimary.Travel.CurrentDirection=cDirectionReverse) AND (lTravelThrottle<0.0))));
                  
END_GET
END_PROPERTY

PROPERTY SteerModeOnFinishing : t_steer_mode
GET
                    SteerModeOnFinishing := lSteerModeOnFinishing;
                  
END_GET
SET
                    lSteerModeOnFinishing := SteerModeOnFinishing;
                  
END_SET
END_PROPERTY

PROPERTY SteerModeRequired : t_steer_mode
GET
                    SteerModeRequired := lSteerModeRequired;
                  
END_GET
SET
                    lSteerModeRequired := SteerModeRequired;
                  
END_SET
END_PROPERTY

PROPERTY TargetAngle : REAL
GET
                    TargetAngle := lTargetAngle;
                  
END_GET
SET
                    lTargetAngle := TargetAngle;
                  
END_SET
END_PROPERTY

PROPERTY TargetAngleIncrement : REAL
GET
                    TargetAngleIncrement := lTargetAngleIncrement;
                  
END_GET
SET
                    lTargetAngleIncrement := TargetAngleIncrement;
                  
END_SET
END_PROPERTY

PROPERTY TargetAngleZeroThreshold : REAL
GET
                    TargetAngleZeroThreshold := lTargetAngleZeroThreshold;
                  
END_GET
SET
                    lTargetAngleZeroThreshold := TargetAngleZeroThreshold;
                  
END_SET
END_PROPERTY

PROPERTY TravelThrottle : t_percentage
GET
                    TravelThrottle := lTravelThrottle;
                  
END_GET
SET
                    lTravelThrottle := TravelThrottle;
                  
END_SET
END_PROPERTY

PROPERTY TypeToken : t_medium_string
GET
                    TypeToken := 'mProgTurn';
                  
END_GET
END_PROPERTY
END_FUNCTION_BLOCK

FUNCTION equalsOperatorWheelAngle : BOOL
  VAR_INPUT
    lAngle1 : REAL;
    lAngle2 : REAL;
    lPrecision : REAL;
  END_VAR

            equalsOperatorWheelAngle := (ABS(lAngle1-lAngle2)<lPrecision);
          
END_FUNCTION

FUNCTION_BLOCK SteerMode EXTENDS NonOperationalParticleSet
  VAR
    lVROverrideReady : ValueReferenceBool;
    lOverrideReady : BOOL := FALSE;
    lEnabled : BOOL := FALSE;
    lAvailable : BOOL := FALSE;
    lSteerAngleMinimum : REAL;
    lSteerAngleMaximum : REAL;
    lTravelThrottleThreshold : t_percentage;
    lMode : t_steer_mode := cSteerModeNone;
  END_VAR

            ;
          

METHOD calculateTravelThrottleThreshold
  VAR_INPUT
    inputAngle : REAL;
  END_VAR
                  
                
END_METHOD

METHOD calculateWheelTargetAngle : t_slew_state
  VAR_INPUT
    wheel : REFERENCE TO SlewMovement;
    inputAngle : REAL;
    steerWheelBase : REAL;
    steerWheelTrack : REAL;
    steerInput : REAL;
  END_VAR
                  calculateWheelTargetAngle.targetAngle := 0.0;
calculateWheelTargetAngle.wheelVelocityFactor := 1.0;
calculateWheelTargetAngle.steerInput := steerInput;
                
END_METHOD

METHOD getInitialTargetAngle : REAL
  VAR_INPUT
    targetAngle : REAL;
    steerMode : t_steer_mode;
  END_VAR
                  getInitialTargetAngle := targetAngle;


                
END_METHOD

METHOD initialize
                  lVROverrideReady.initializeValueReference(lOverrideReady,NopSelf,'OvrdReady','Override ready checks','',cValueStyleParameter);

SUPER^.initialize();

lSteerAngleMinimum := gSystemPrimary.Steering.SteerAnglePhysicalMinimum;
lSteerAngleMaximum := gSystemPrimary.Steering.SteerAnglePhysicalMaximum;
lTravelThrottleThreshold := 1.0;

                
END_METHOD

METHOD leave
                  
                
END_METHOD

METHOD matches : BOOL
  VAR_INPUT
    steerMode : t_steer_mode;
  END_VAR
                  matches := (steerMode=lMode);
                
END_METHOD

METHOD ready : BOOL
  VAR_INPUT
    state : t_adjust_state;
  END_VAR
                  ready := ((state<cAdjustStateAdjusting) OR
	(lOverrideReady));

                
END_METHOD

PROPERTY Available : BOOL
GET
                    Available := lAvailable;
                  
END_GET
SET
                    lAvailable := Available;
                  
END_SET
END_PROPERTY

PROPERTY Enabled : BOOL
GET
                    Enabled := ((lEnabled) and (lAvailable));
                  
END_GET
SET
                    lEnabled := Enabled;
                  
END_SET
END_PROPERTY

PROPERTY Mode : t_steer_mode
GET
                    Mode := lMode;
                  
END_GET
END_PROPERTY

PROPERTY SteerAngleMaximum : REAL
GET
                    SteerAngleMaximum := lSteerAngleMaximum;
                  
END_GET
END_PROPERTY

PROPERTY SteerAngleMinimum : REAL
GET
                    SteerAngleMinimum := lSteerAngleMinimum;
                  
END_GET
END_PROPERTY

PROPERTY TravelThrottleThreshold : t_percentage
GET
                    TravelThrottleThreshold := lTravelThrottleThreshold;
                  
END_GET
END_PROPERTY

PROPERTY TypeToken : t_medium_string
GET
                    TypeToken := 'SteerMode';
                  
END_GET
END_PROPERTY
END_FUNCTION_BLOCK

FUNCTION_BLOCK SteerMode4WS EXTENDS SteerMode
  VAR CONSTANT
    cSteerAngleMinimum : REAL := ((-45.0 / 180.0) * cPi);
    cSteerAngleMaximum : REAL := ((45.0 / 180.0) * cPi);
    cTravelThresholdUnrestrictedAngle : REAL := (cSteerAngleMaximum * 0.5);
    cTravelThresholdMinimumThreshold : REAL := 0.3;
  END_VAR
  VAR
    lTravelThresholdFactor : REAL := 0.0;
  END_VAR

            ;
          

METHOD calculateTravelThrottleThreshold
  VAR_INPUT
    inputAngle : REAL;
  END_VAR
                  IF (ABS(inputAngle)<cTravelThresholdUnrestrictedAngle) THEN
	lTravelThrottleThreshold := 1.0;
	RETURN;
END_IF

lTravelThrottleThreshold := ABS(1.0 + (ABS(inputAngle)-cTravelThresholdUnrestrictedAngle)*lTravelThresholdFactor);


                
END_METHOD

METHOD calculateWheelTargetAngle : t_slew_state
  VAR_INPUT
    wheel : REFERENCE TO SlewMovement;
    inputAngle : REAL;
    steerWheelBase : REAL;
    steerWheelTrack : REAL;
    steerInput : REAL;
  END_VAR
  VAR
    tmpReal : REAL;
    targetAngle : REAL;
    wheelVelocityFactor : REAL;
    steerAngleOuter : REAL;
  END_VAR
                  (* 4WS
	lSteerAngle = alpha
	lSteerAngleOuter = beta = arctan( B*TAN(alpha) / (B+2T*TAN(alpha)))	*)

tmpReal := TAN(ABS(inputAngle));
steerAngleOuter := ATAN(steerWheelBase * tmpReal /
		(steerWheelBase + 2.0 * tmpReal * steerWheelTrack));

IF (inputAngle=0) THEN
	wheelVelocityFactor := 1.0;
	targetAngle := 0;
	
ELSIF ((wheel.InnerFlag) XOR (inputAngle>0)) THEN
	(* the outer wheel
		~inner on positive angles
		inner on negative angles *)
	targetAngle := wheel.StandardSign * steerAngleOuter * inputAngle/ABS(inputAngle);

	(* outer wheel is at requested speed *)
	wheelVelocityFactor := 1.0;

ELSE
	(* the inner wheel
		inner on positive angles
		~inner on negative angles *)
	targetAngle := wheel.StandardSign * inputAngle;

	(* single wheel per yoke: ratio of inner/outer = SIN(beta)/SIN(alpha)
	lWheelVelocityFactor := SIN(lSteerAngleOuter)/SIN(ABS(lSteerAngle)); *)

	(* ratio of inner/outer = [B/(2.SIN(alpha)) - offset]/[B/(2.SIN(beta)) + offset] *)
	wheelVelocityFactor := (steerWheelBase/(2*SIN(ABS(inputAngle))))/
		(steerWheelBase/(2*SIN(ABS(steerAngleOuter))));
END_IF

calculateWheeltargetAngle.targetAngle := targetAngle;
calculateWheeltargetAngle.wheelVelocityFactor := wheelVelocityFactor;
calculateWheeltargetAngle.steerInput := steerInput * wheel.StandardSign;

                
END_METHOD

METHOD initialize
                  Name := 'Steer4WS';
SUPER^.initialize();

lMode := cSteerMode4WS;
	
lSteerAngleMinimum := cSteerAngleMinimum;
lSteerAngleMaximum := cSteerAngleMaximum;

lTravelThresholdFactor := (1.0-cTravelThresholdMinimumThreshold)/(cTravelThresholdUnrestrictedAngle-cSteerAngleMaximum);


                
END_METHOD
END_FUNCTION_BLOCK

FUNCTION_BLOCK SteerModeCarousel EXTENDS SteerMode
  VAR CONSTANT
    cTravelThrottleThreshold : t_percentage := 0.25;
  END_VAR

            ;
          

METHOD calculateWheelTargetAngle : t_slew_state
  VAR_INPUT
    wheel : REFERENCE TO SlewMovement;
    inputAngle : REAL;
    steerWheelBase : REAL;
    steerWheelTrack : REAL;
    steerInput : REAL;
  END_VAR
  VAR
    targetAngle : REAL;
    wheelVelocityFactor : REAL;
  END_VAR
                  targetAngle := gSystemPrimary.Steering.CarouselAngle * wheel.CarouselSign;

IF (wheel.IndependentWheels) THEN
	IF (wheel.InnerFlag) THEN
		wheelVelocityFactor := -1.0;
	ELSE
		wheelVelocityFactor := 1.0;
	END_IF
ELSE
	wheelVelocityFactor := 1.0;
	
	IF ((wheel.DriveWheel) AND (wheel.InnerFlag)) THEN
		targetAngle := targetAngle - 3.14159265;
	END_IF
END_IF

calculateWheeltargetAngle.targetAngle := targetAngle;
calculateWheeltargetAngle.wheelVelocityFactor := wheelVelocityFactor;
calculateWheeltargetAngle.steerInput := 0.0;

                
END_METHOD

METHOD initialize
                  Name := 'SteerCarousel';
SUPER^.initialize();

lMode := cSteerModeCarousel;

lTravelThrottleThreshold := cTravelThrottleThreshold;

                
END_METHOD
END_FUNCTION_BLOCK

FUNCTION_BLOCK SteerModeCustom EXTENDS SteerMode
  VAR CONSTANT
    cTravelThrottleThreshold : t_percentage := 0.0;
    cTargetAngleA : REAL := 0.0;
    cTargetAngleB : REAL := cPi;
    cTargetAngleC : REAL := 0.0;
    cTargetAngleD : REAL := cPi;
  END_VAR

            ;
          

METHOD calculateWheelTargetAngle : t_slew_state
  VAR_INPUT
    wheel : REFERENCE TO SlewMovement;
    inputAngle : REAL;
    steerWheelBase : REAL;
    steerWheelTrack : REAL;
    steerInput : REAL;
  END_VAR
                  CASE wheel.ID OF
	1:
		calculateWheeltargetAngle.targetAngle := cTargetAngleA;
	
	2:
		calculateWheeltargetAngle.targetAngle := cTargetAngleB;

	3:
		calculateWheeltargetAngle.targetAngle := cTargetAngleC;

	4:
		calculateWheeltargetAngle.targetAngle := cTargetAngleD;
END_CASE

calculateWheeltargetAngle.wheelVelocityFactor := 0.0;
calculateWheeltargetAngle.steerInput := 0.0;



                
END_METHOD

METHOD initialize
                  Name := 'SteerCustom';
SUPER^.initialize();

lMode := cSteerModeCustom;

lTravelThrottleThreshold := cTravelThrottleThreshold;

                
END_METHOD
END_FUNCTION_BLOCK

FUNCTION_BLOCK SteerModeLateral EXTENDS SteerMode
  VAR CONSTANT
    cTravelThrottleThreshold : t_percentage := 0.35;
    cSteerAngleMinimum : REAL := ((-92.0 / 180.0) * cPi);
    cSteerAngleMaximum : REAL := ((92.0 / 180.0) * cPi);
  END_VAR

            ;
          

METHOD calculateWheelTargetAngle : t_slew_state
  VAR_INPUT
    wheel : REFERENCE TO SlewMovement;
    inputAngle : REAL;
    steerWheelBase : REAL;
    steerWheelTrack : REAL;
    steerInput : REAL;
  END_VAR
                  calculateWheeltargetAngle.targetAngle := inputAngle;
calculateWheeltargetAngle.wheelVelocityFactor := 1.0;
calculateWheeltargetAngle.steerInput := steerInput;

                
END_METHOD

METHOD getInitialTargetAngle : REAL
  VAR_INPUT
    targetAngle : REAL;
    steerMode : t_steer_mode;
  END_VAR
                  IF (steerMode=cSteerModeLateralNeg90) THEN
	getInitialTargetAngle := -cPiOn2;
ELSIF (steerMode=cSteerModeLateralPos90) THEN
	getInitialTargetAngle := cPiOn2;
ELSE	
	getInitialTargetAngle := 0.0;
END_IF


                
END_METHOD

METHOD initialize
                  Name := 'SteerLateral';
SUPER^.initialize();

lMode := cSteerModeLateral;

lTravelThrottleThreshold := cTravelThrottleThreshold;

lSteerAngleMinimum := cSteerAngleMinimum;
lSteerAngleMaximum := cSteerAngleMaximum;
                
END_METHOD

METHOD matches : BOOL
  VAR_INPUT
    steerMode : t_steer_mode;
  END_VAR
                  matches := ((steerMode=lMode) OR
	(steerMode=cSteerModeLateralNeg90) OR
	(steerMode=cSteerModeLateralPos90));

                
END_METHOD
END_FUNCTION_BLOCK

FUNCTION_BLOCK SteerModeReconfigure EXTENDS SteerMode
  VAR CONSTANT
    cTravelThrottleThreshold : t_percentage := 0.5;
  END_VAR

            ;
          

METHOD calculateWheelTargetAngle : t_slew_state
  VAR_INPUT
    wheel : REFERENCE TO SlewMovement;
    inputAngle : REAL;
    steerWheelBase : REAL;
    steerWheelTrack : REAL;
    steerInput : REAL;
  END_VAR
                  // positive is extension, wheelD is reversed, wheelC is normal
IF ((wheel.DriveWheel) AND (NOT(wheel.InnerFlag))) THEN
	calculateWheelTargetAngle.targetAngle := 0.0 - cPIOn2;
ELSE
	calculateWheelTargetAngle.targetAngle := cPIOn2;
END_IF

calculateWheelTargetAngle.wheelVelocityFactor := 1.0;
calculateWheeltargetAngle.steerInput := 0.0;

                
END_METHOD

METHOD initialize
                  Name := 'SteerReconfigure';
SUPER^.initialize();

lMode := cSteerModeReconfigure;

lTravelThrottleThreshold := cTravelThrottleThreshold;
                
END_METHOD

METHOD leave
                  lEnabled := false;
                
END_METHOD

METHOD ready : BOOL
  VAR_INPUT
    state : t_adjust_state;
  END_VAR
                  ready := ((state=cAdjustStateGood) OR
	(lOverrideReady));

                
END_METHOD
END_FUNCTION_BLOCK

FUNCTION_BLOCK SlewMovement EXTENDS CheckedMovement
  VAR
    cSteerDeltaZeroThreshold : REAL := 0.015;  (* implies min throttle ( * increased from 0.010 from 0.005 from 0.0025 * ) *)
    cSteerDeltaZeroThresholdChangingMode : REAL := 0.025;
    cSteerDeltaZeroThresholdMax : REAL := 0.03;
    cSteerDeltaZeroThresholdGain : REAL := 0.002;
    cTargetAngleAdjustment : REAL := 0.01;
    cDeltaConvergingRestartThreshold : REAL := 0.02;
    cRequestedEquivalentThreshold : REAL := 0.001;
    cDeltaCancelMovementCount : USINT := 2;
    cSteerVelocityZeroThreshold : REAL := 0.1;
    cSteerThrottleFactor : REAL := -14.0;  (* max throttle of 0.54, increased from -6.0 to -7.0 for elextric, up to -14 for hydraulic m190 * ) *)
    cSteerAngleMaxSensorDelta : REAL := 0.3;  (* Up from 0.1 *)
    cSteerAngleMaxDelta : REAL := 0.06;  (* implies max throttle, limits magnitude of correction, should not saturate the drive *)
    cSteerAngleMaxErrorDelta : REAL := 0.15;  (* limit on when to halt the system, increase from 0.1, control should be stable 99.9999% of the time under normal operation *)
    cSteerAngleMaxMovementDelta : REAL := 0.5;
    cSteerMovementCountMax : UINT := 3;
    cControlSystemKp : REAL := 14.0;
    cControlSystemKi : REAL := 40.0;
    cControlSystemKd : REAL := 0.0;
    cThrottleMax : REAL := 0.8;
    cTargetStationaryPeriod : t_time := TIME#1s0ms;
    cOvershootPeriod : t_time := TIME#500ms;
    cTargetAngleChangeThreshold : REAL := 0.01;
    cMovementCountOvershoot : USINT := 1;
    lVROverideControl : ValueReferenceBool;
    lOverideControl : BOOL := FALSE;
    lVREnableMovementManagement : ValueReferenceBool;
    lEnableMovementManagement : BOOL := TRUE;
    lVREnableOvershoot : ValueReferenceBool;
    lEnableOvershoot : BOOL := TRUE;
    lVREnableTargetPrediction : ValueReferenceBool;
    lEnableTargetPrediction : BOOL := TRUE;
    lVREnableModeChangeClearOnOK : ValueReferenceBool;
    lEnableModeChangeClearOnOK : BOOL := TRUE;
    lAlarmSteerLargeSensorDelta : ReportableAlarm;  (* foobar *)
    lControllerSteerAngle : REFERENCE TO ControllerRotaryEncoderRange;
    lSteerMovement : REFERENCE TO SteerMovement;
    lTravelMovement : REFERENCE TO Movement;
    lID : BYTE := 0;  (* lControllerIO: REFERENCE TO ControllerIO; lControllerMotor: REFERENCE TO ControllerMotor; lControlSystem: PID; *)
    lCarouselSign : REAL;
    lStandardSign : REAL;
    lInnerFlag : BOOL;
    lDriveWheel : BOOL := TRUE;
    lIndependentWheels : BOOL := FALSE;
    lSteerInput : REAL;
    lCurrentVelocity : REAL;
    lCurrentAngle : REAL;
    lPreviousAngle : REAL;
    lTargetAngle : REAL;
    lTargetPredictionOffset : REAL;
    lPredictedTargetAngle : REAL;
    lPreviousTargetAngle : REAL;
    lTargetAngleAdjusted : REAL;
    lTargetAngleAdjustment : REAL := 0.0;
    lDelta : REAL;
    lFilteredDelta : REAL;
    lDeltaPrevious : REAL;
    lDeltaConverging : BOOL := FALSE;
    lControlFeedbackSign : REAL := 1.0;
    lThrottleMinThreshold : REAL := 0.0;
    lWheelVelocityFactor : REAL;
    lWheelDirection : REAL;
    lRequested : t_percentage := 0.0;
    lRequestedCurve : ValueObjectPercentageCurve;
    lRequestedPID : t_percentage;  (* lRequestedPrevious: t_percentage:= 0.0; lRequestedNonZero: t_percentage:= 0.0; lRequestedNonZeroPrevious: t_percentage:= 0.0; lRequestedDelta: t_percentage:= 0.0; lRequestedDeltaPrevious: t_percentage:= 0.0; *)
    lRequestedSimple : t_percentage;
    lRequestDelta : t_percentage;
    lEnableControlSystem : BOOL := FALSE;
    lDeltaZeroThreshold : REAL := cSteerDeltaZeroThreshold;
    lModeChange : BOOL := FALSE;
    lModeChangeDisableControl : BOOL := FALSE;
    lState : t_adjust_state := cAdjustStateNone;
    lMovementCount : UINT;
    lMovementEventCount : UINT := 0;
    lTargetStationary : BOOL;
    lTargetStationaryTimer : t_timer;
    lOvershoot : BOOL;
    lOvershootTimer : t_timer;
  END_VAR

            ;
          

METHOD checkWheelState
                  IF (ABS(lCurrentVelocity)<cSteerVelocityZeroThreshold) THEN
	lCurrentVelocity := 0;
END_IF

IF  (ABS(lCurrentAngle-lPreviousAngle) >= cSteerAngleMaxSensorDelta) THEN
	lAlarmSteerLargeSensorDelta.report(FALSE); //foobar
END_IF

lPredictedTargetAngle := lTargetAngle;
lTargetPredictionOffset := 0.0;
IF (lEnableTargetPrediction) THEN
	IF ((lSteerInput>0.0) AND
		(lCurrentAngle>lTargetAngle)) THEN
		lPredictedTargetAngle := lCurrentAngle;
		lTargetPredictionOffset := lPredictedTargetAngle - lTargetAngle;
	END_IF
	IF ((lSteerInput<0.0) AND
		(lCurrentAngle<lTargetAngle)) THEN
		lPredictedTargetAngle := lCurrentAngle;
		lTargetPredictionOffset := lPredictedTargetAngle - lTargetAngle;
	END_IF
END_IF

IF (lOverideControl) THEN
	lCurrentVelocity := 0;
	lTargetAngleAdjustment := 0.0;
	lDeltaConverging := FALSE;
	lPreviousAngle := lCurrentAngle := lTargetAngleAdjusted := lPredictedTargetAngle := lTargetAngle;
END_IF

lDeltaPrevious := lDelta;
lDelta := (lCurrentAngle-lTargetAngle) * lControlFeedbackSign;
lState := cAdjustStateAdjusting;

IF (ABS(lDelta)>=cSteerAngleMaxErrorDelta) THEN
	lState := cAdjustStateError;
END_IF

IF (ABS(lDelta)>cDeltaConvergingRestartThreshold) THEN
	lDeltaConverging := TRUE;
	lTargetAngleAdjustment := cTargetAngleAdjustment;
END_IF

IF (Stationary) THEN
	lDeltaConverging := FALSE;
END_IF

IF (lMovementCount>=cDeltaCancelMovementCount) THEN
	lDeltaConverging := FALSE;	
END_IF

lDeltaConverging := (((lDeltaPrevious*lDelta) > 0.0) AND
	(lDeltaConverging));;

IF ((NOT(lDeltaConverging)) OR
	(lTravelMovement.InputPresentAny))  THEN
	lTargetAngleAdjustment := 0.0;
END_IF

IF (lCurrentAngle<lPredictedTargetAngle) THEN
	lTargetAngleAdjusted := lPredictedTargetAngle + lTargetAngleAdjustment;
ELSIF (lCurrentAngle>lPredictedTargetAngle) THEN
	lTargetAngleAdjusted := lPredictedTargetAngle - lTargetAngleAdjustment;
ELSE
	lTargetAngleAdjusted := lPredictedTargetAngle;
END_IF

IF (lTargetAngleAdjusted>lSteerMovement.SteerAngleMaximum) THEN
	lTargetAngleAdjusted := lSteerMovement.SteerAngleMaximum;
END_IF
IF (lTargetAngleAdjusted<lSteerMovement.SteerAngleMinimum) THEN
	lTargetAngleAdjusted := lSteerMovement.SteerAngleMinimum;
END_IF

lFilteredDelta := (lCurrentAngle-lTargetAngleAdjusted) * lControlFeedbackSign;

IF (ABS(lFilteredDelta)>=cSteerAngleMaxDelta) THEN
	lFilteredDelta := cSteerAngleMaxDelta * lFilteredDelta/ABS(lFilteredDelta);
END_IF

IF (lEnableOvershoot) THEN
	lOvershoot := ((lMovementCount>=cMovementCountOvershoot) AND
		(NOT(lTravelMovement.InputPresentAny)));

	IF (lOvershoot) THEN
		lFilteredDelta := 0.0;
	END_IF

(*	IF (lOvershoot) THEN
		lOvershootTimer.operator();

		IF (NOT(lOvershootTimer.Expired)) THEN
			lFilteredDelta := 0.0;
		END_IF
	ELSE
		lOvershootTimer.reset();	
	END_IF*)
END_IF

IF (ABS(lDelta)<lDeltaZeroThreshold) THEN
	IF (Stationary) THEN
		lModeChange := FALSE;
		lDeltaZeroThreshold := cSteerDeltaZeroThreshold;
	END_IF
	
	IF (NOT(lDeltaConverging)) THEN
		lState :=cAdjustStateGood;
		lFilteredDelta := 0;
		lTargetAngleAdjustment := 0.0;
	END_IF
END_IF

IF ((lModeChange) AND
	(OK) AND
	(lEnableModeChangeClearOnOK)) THEN
	lModeChange := FALSE;
END_IF

lRequestedSimple := lFilteredDelta*cSteerThrottleFactor;

(*lControlSystem.KP := cControlSystemKp;
lControlSystem.TN := cControlSystemKi;
lControlSystem.TV := cControlSystemKd;
lControlSystem.Y_OFFSET := 0;
lControlSystem.Y_MAX := cThrottleMax;
lControlSystem.Y_MIN := -1.0 * cThrottleMax;

lControlSystem.SET_POINT := lTargetAngleAdjusted;
lControlSystem.ACTUAL := lCurrentAngle;
lControlSystem.RESET := FALSE;

lControlSystem();

//lControlSystem.LIMITS_ACTIVE
//lControlSystem.OVERFLOW
lRequestedPID := lControlSystem.Y * lControlFeedbackSign;

IF (lEnableControlSystem) THEN
	lRequested := lRequestedPID;
ELSE
	lRequested := lRequestedSimple;
END_IF*)
lRequested := lRequestedSimple;

lRequestDelta := lRequestedPID - lRequestedSimple;

                
END_METHOD

METHOD hunting
                  
(*lRequestedDeltaPrevious := lRequestedDelta;
IF (ABS(lRequested-lRequestedPrevious)>=cRequestedEquivalentThreshold) THEN
	lRequestedDelta := lRequested - lRequestedPrevious;
END_IF

lRequestedNonZeroPrevious := lRequestedNonZero;
IF (ABS(lRequested)>=cRequestedEquivalentThreshold) THEN
	lRequestedNonZero := lRequested;
END_IF*)

IF ((ABS(lCurrentAngle-lPreviousAngle) >= cSteerAngleMaxMovementDelta) OR
	(ABS(lTargetAngle-lPreviousTargetAngle)>cTargetAngleChangeThreshold) OR
	(lTravelMovement.InputPresentAny) OR
	(lSteerMovement.InputPresentAny) OR
	(gSystemPrimary.SystemState.State<cSystemStateOperational)) THEN
	lRequestedCurve.reset();
	
	//lMovementCount := 0;
	//lRequestedDelta := 0.0;
	//lRequestedDeltaPrevious := 0.0;
END_IF

lRequestedCurve.InputAsPercentage := lRequested;
lRequestedCurve.operator();
lMovementCount := lRequestedCurve.Inflexions;

(*IF (((lRequestedDeltaPrevious<0.0) AND (lRequestedDelta>0.0)) OR
	((lRequestedDeltaPrevious>0.0) AND (lRequestedDelta<0.0)) OR
	((lRequestedNonZeroPrevious<0.0) AND (lRequestedNonZero>0.0)) OR
	((lRequestedNonZeroPrevious>0.0) AND (lRequestedNonZero<0.0))) THEN
	lMovementCount := lMovementCount + 1;
	IF (lMovementCount>cSteerMovementCountMax) THEN
		lMovementEventCount := lMovementEventCount + 1;
	END_IF
END_IF*)

(*IF (((lRequestedPrevious=0.0) AND (lRequested<>0.0)) OR}
	((lRequestedPrevious<0.0) AND (lRequested>0.0)) OR
	((lRequestedPrevious>0.0) AND (lRequested<0.0))) THEN
	lMovementCount := lMovementCount + 1;
	IF (lMovementCount>cSteerMovementCountMax) THEN
		lMovementEventCount := lMovementEventCount + 1;
	END_IF
END_IF *)

IF ((lEnableMovementManagement) AND (lMovementCount>cSteerMovementCountMax)) THEN
	lRequested := 0.0;
	Diagnostic := cMovementDiagnosticHunting;
END_IF
                
END_METHOD

METHOD initialize
                  IF ((NOT(__ISVALIDREF(lThrottle))) OR
	(NOT(__ISVALIDREF(lControllerSteerAngle))) OR
	(NOT(__ISVALIDREF(lSteerMovement))) OR
	(NOT(__ISVALIDREF(lTravelMovement)))) THEN
	gCodeErrorHandler(pMessage:=CONCAT('null reference in ',lIdentity));
END_IF

lVROverideControl.initializeValueReference(lOverideControl,NopSelf,'OverrideControl','Disable automatic control','',cValueStyleParameter);

lVREnableMovementManagement.initializeValueReference(lEnableMovementManagement,NopSelf,'EnblMovMgmt','Enable movement management','',cValueStyleParameter);
lVREnableOvershoot.initializeValueReference(lEnableOvershoot,NopSelf,'EnblOvershoot','Enable overshoot control','',cValueStyleParameter);
lVREnableTargetPrediction.initializeValueReference(lEnableTargetPrediction,NopSelf,'EnblPrediction','Enable predictive control','',cValueStyleParameter);
lVREnableModeChangeClearOnOK.initializeValueReference(lEnableModeChangeClearOnOK,NopSelf,'EnblMdChngClr','Enable mode change clear on OK','',cValueStyleParameter);
	
lAlarmSteerLargeSensorDelta.initializeState(NopSelf,'',cACSteerALargeSensorDelta);

lRequestedCurve.initializeValueObject(NopSelf,'Curve','Control curve metric','',cValueStyleConfigurable);

SUPER^.initialize();

lFunctionalMode := cFunctionalModeAny;

lRegisterUMFSPrimary := FALSE;
lRegisterUMFSAuxilliary := FALSE;
lRegisterUMFSSecondary := FALSE;

lRegisterActive := FALSE;
lRegisterOperatingMode := FALSE;
	
lEnabled := TRUE;
lEnableOperatingModeSlow := FALSE;
lEnableOnlyOnActiveAllow := FALSE;
lEnableUMFSCheck := FALSE;

cSteerDeltaZeroThreshold := 0.015; // implies min throttle (* increased from 0.010 from 0.005 from 0.0025 *)
cSteerDeltaZeroThresholdChangingMode := 0.025;
cSteerDeltaZeroThresholdMax := 0.030;
cSteerDeltaZeroThresholdGain := 0.002;
cTargetAngleAdjustment := 0.0;
cDeltaConvergingRestartThreshold := 0.015;
cRequestedEquivalentThreshold := 0.05;
cDeltaCancelMovementCount := 1;
	
cSteerVelocityZeroThreshold := 0.1;
cSteerThrottleFactor := -8.0; // max throttle of 0.54, increased from -6.0 to -7.0 up to -10.0 down to -8.0 for elextric, up to -14 for hydraulic m190 *)
cSteerAngleMaxSensorDelta := 0.3; (* Up from 0.1 *)
cSteerAngleMaxDelta := 0.08; // implies max throttle, limits magnitude of correction, should not saturate the drive
cSteerAngleMaxErrorDelta := 0.15; // limit on when to halt the system
cSteerAngleMaxMovementDelta := 0.5;

cSteerMovementCountMax := 3;

cControlSystemKp := 14.0;
cControlSystemKi := 40.0;
cControlSystemKd := 0.0;
cThrottleMax := 0.8;	
	
cTargetStationaryPeriod := T#1S;
cOvershootPeriod := T#500MS;
cTargetAngleChangeThreshold := 0.01;
cMovementCountOvershoot := 1;

(*lControlSystem.KP := cControlSystemKp;
lControlSystem.TN := cControlSystemKi;
lControlSystem.TV := cControlSystemKd;
lControlSystem.Y_OFFSET := 0;
lControlSystem.Y_MAX := cThrottleMax;
lControlSystem.Y_MIN := -1.0 * cThrottleMax;
lControlSystem.RESET := TRUE;
lControlSystem();
lControlSystem.RESET := FALSE;*)

lTargetStationaryTimer.initialize();
lTargetStationaryTimer.Enable := TRUE;
lTargetStationaryTimer.Period := cTargetStationaryPeriod;

lOvershootTimer.initialize();
lOvershootTimer.Enable := TRUE;
lOvershootTimer.Period := cOvershootPeriod;




                
END_METHOD

METHOD operator
                  // angle in radians
lPreviousAngle := lCurrentAngle;
lPreviousTargetAngle := lTargetAngle;
//lRequestedPrevious := lRequested;

IF (lTargetAngle<>lPreviousTargetAngle) THEN
	lTargetStationaryTimer.reset();
END_IF
lTargetStationaryTimer.operator();
lTargetStationary := lTargetStationaryTimer.Expired;

lCurrentAngle := lControllerSteerAngle.Angle;

// velocity in hz
lCurrentVelocity := lControllerSteerAngle.AngularVelocity;

checkWheelState();

lEnableUMFSCheck := NOT(ModeChange);

IF ((lRequested<>0.0) AND
	(ABS(lRequested)<lThrottleMinThreshold)) THEN
	lRequested := lThrottleMinThreshold*lRequested/ABS(lRequested);
END_IF

hunting();

IF (lModeChangeDisableControl) THEN
	lRequested := 0.0;
END_IF

lInput.InputAsPercentage := lRequested;
lInput.operator();

SUPER^.operator();

                
END_METHOD

METHOD initializeSlew
  VAR_INPUT
    throttle : REFERENCE TO Throttle;
    controller : REFERENCE TO ControllerRotaryEncoderRange;
    steerMovement : REFERENCE TO SteerMovement;
    travelMovement : REFERENCE TO Movement;
  END_VAR
                  lThrottle REF= throttle;
lControllerSteerAngle REF= controller;
lSteerMovement REF= steerMovement;
lTravelMovement REF= travelMovement;

                
END_METHOD

PROPERTY CarouselSign : REAL
GET
                    CarouselSign := lCarouselSign;
                  
END_GET
SET
                    lCarouselSign := CarouselSign;
                  
END_SET
END_PROPERTY

PROPERTY ControlFeedbackSign : REAL
GET
                    ControlFeedbackSign := lControlFeedbackSign;
                  
END_GET
SET
                    lControlFeedbackSign := ControlFeedbackSign;
                  
END_SET
END_PROPERTY

PROPERTY ControllerSteerAngle : REFERENCE TO ControllerRotaryEncoderRange
GET
                    ControllerSteerAngle ref= lControllerSteerAngle; // foobar remove property?
                  
END_GET
END_PROPERTY

PROPERTY CurrentAngle : REAL
GET
                    CurrentAngle := lCurrentAngle;
                  
END_GET
END_PROPERTY

PROPERTY CurrentVelocity : REAL
GET
                    CurrentVelocity := lCurrentVelocity;
                  
END_GET
END_PROPERTY

PROPERTY Delta : REAL
GET
                    Delta := lDelta;
                  
END_GET
END_PROPERTY

PROPERTY DriveWheel : BOOL
GET
                    DriveWheel := lDriveWheel;
                  
END_GET
SET
                    lDriveWheel := DriveWheel;
                  
END_SET
END_PROPERTY

(* {attribute 'monitoring' := 'call'} *)
PROPERTY FilteredDelta : REAL
GET
                    FilteredDelta := lFilteredDelta;
                  
END_GET
END_PROPERTY

PROPERTY ID : BYTE
GET
                    ID := lID;
                  
END_GET
SET
                    lID := ID;
                  
END_SET
END_PROPERTY

PROPERTY IndependentWheels : BOOL
GET
                    IndependentWheels := lIndependentWheels;
                  
END_GET
SET
                    lIndependentWheels := IndependentWheels;
                  
END_SET
END_PROPERTY

PROPERTY InnerFlag : BOOL
GET
                    InnerFlag := lInnerFlag;
                  
END_GET
SET
                    lInnerFlag := InnerFlag;
                  
END_SET
END_PROPERTY

PROPERTY ModeChange : BOOL
GET
                    ModeChange := lModeChange;
                  
END_GET
SET
                    lModeChange := ModeChange;

IF (lModeChange) THEN
	lDeltaZeroThreshold := cSteerDeltaZeroThresholdChangingMode;
ELSE
	lDeltaZeroThreshold := cSteerDeltaZeroThreshold;
END_IF

                  
END_SET
END_PROPERTY

PROPERTY ModeChangeDisableControl : BOOL
GET
                    ModeChangeDisableControl := lModeChangeDisableControl;
                  
END_GET
SET
                    lModeChangeDisableControl := ModeChangeDisableControl;

                  
END_SET
END_PROPERTY

(* {attribute 'monitoring' := 'call'} *)
PROPERTY OK : BOOL
GET
                    OK := ((lState>=cAdjustStateGood) OR
	(lState<=cAdjustStateAdjusting));
                  
END_GET
END_PROPERTY

PROPERTY StandardSign : REAL
GET
                    StandardSign := lStandardSign;
                  
END_GET
SET
                    lStandardSign := StandardSign;
                  
END_SET
END_PROPERTY

(* {attribute 'monitoring' := 'call'} *)
PROPERTY State : t_adjust_state
GET
                    State := lState;

                  
END_GET
END_PROPERTY

PROPERTY Target : t_slew_state
SET
                    lTargetAngle := Target.targetAngle;
lWheelVelocityFactor := Target.wheelVelocityFactor;
lSteerInput := Target.steerInput;
                  
END_SET
END_PROPERTY

PROPERTY TargetAngle : REAL
GET
                    TargetAngle := lTargetAngle;

                  
END_GET
END_PROPERTY

PROPERTY ThrottleMinThreshold : REAL
GET
                    ThrottleMinThreshold := lThrottleMinThreshold;
                  
END_GET
SET
                    lThrottleMinThreshold := ThrottleMinThreshold;
                  
END_SET
END_PROPERTY

PROPERTY TypeToken : t_medium_string
GET
                    TypeToken := 'mSlew';
                  
END_GET
END_PROPERTY

PROPERTY WheelDirection : REAL
GET
                    WheelDirection := lWheelDirection;
                  
END_GET
SET
                    lWheelDirection := WheelDirection;
                  
END_SET
END_PROPERTY

PROPERTY WheelVelocityFactor : REAL
GET
                    WheelVelocityFactor := lWheelVelocityFactor;
                  
END_GET
END_PROPERTY
END_FUNCTION_BLOCK

FUNCTION_BLOCK SteerMovement EXTENDS CheckedMovement
  VAR CONSTANT
    cSteerAnglePhysicalMinimum : REAL := ((-184.0 / 180.0) * cPi);
    cSteerAnglePhysicalMaximum : REAL := ((184.0 / 180.0) * cPi);
    cTargetAngleUpdatePeriod : t_ms_time := TIME#25ms;
    cOperatingModeLockPeriod : t_time := TIME#1s0ms;
  END_VAR
  VAR
    cSteerAngleMaxUpdateDelta : REAL := 0.06;  (* limit on how far away the target can be pushed *)
    cSteerAngleMaxDerivedUpdateDelta : REAL := 0.07;
    cSteerAngleThrottleIncrement : REAL := 0.08;
    cSteerAngleDeltaGain : t_percentage := 1.0;
    cSteerAbsoluteShiftFactor : REAL := 2.0;
    lVREnableRelativeSteering : ValueReferenceBool;
    lEnableRelativeSteering : BOOL := FALSE;
    lVREnableZeroTargetAngleSwitch : ValueReferenceBool;
    lEnableZeroTargetAngleSwitch : BOOL := TRUE;
    lVREnableSequentialModeChange : ValueReferenceBool;
    lEnableSequentialModeChange : BOOL := TRUE;
    lVREnableActiveOnModeChange : ValueReferenceBool;
    lEnableActiveOnModeChange : BOOL := TRUE;
    lVREnableDerivedTargetAngleIncrement : ValueReferenceBool;
    lEnableDerivedTargetAngleIncrement : BOOL := FALSE;
    lVREnableOperatingModeLockOnSteerModeChange : ValueReferenceBool;
    lEnableOperatingModeLockOnSteerModeChange : BOOL := FALSE;
    lEnableUpdateTimer : BOOL := FALSE;
    _Throttle : ThrottleVirtual;
    lWheelA : SlewMovement;
    lWheelB : SlewMovement;
    lWheelC : SlewMovement;
    lWheelD : SlewMovement;
    lSteerMode4WS : SteerMode4WS;
    lSteerModeLateral : SteerModeLateral;
    lSteerModeCarousel : SteerModeCarousel;
    lSteerModeReconfigure : SteerModeReconfigure;
    lSteerModeCustom : SteerModeCustom;
    lMode : REFERENCE TO SteerMode;
    lModeChange : BOOL;
    lAdjustState : t_adjust_state;
    lSteerModeDiagnostic : t_steer_mode_diagnostic;
    lTargetAngle : ValueObjectReal;
    lRequestedAbsoluteTargetAngle : REAL;
    lTargetAngleShift : REAL;
    lTargetAngleIncrement : REAL := 0;
    lTargetAngleIncrementDerived : REAL := 0;
    lTargetAngleIncrementDerivedPost : REAL := 0;
    lTargetAngleUpdateTimer : t_timer;
    lStationaryTargetAngleIncrement : REAL := 0.005;
    lSteerWheelTrack : REAL := 4100.0;
    lSteerWheelBase : REAL := 5000.0;
    lCarouselAngle : REAL;
    lCurrentAbsDelta : REAL;
    lCurrentPositiveDelta : REAL;
    lCurrentNegativeDelta : REAL;
    lStationary : BOOL;
    lStalled : BOOL;
    lStalledSubSystemsPrevious : BOOL;
    lStalledSubSystems : BOOL;
    lStallClearPreCondition : BOOL;
    lStallClearPreConditionCleared : BOOL;
    lZeroTargetAngleSwitch : ValueObjectBool;
  END_VAR

            ;
          

METHOD checkModeEnabled : BOOL
  VAR_INPUT
    mode : t_steer_mode;
  END_VAR
                  checkModeEnabled := getMode(mode).Enabled;

                
END_METHOD

METHOD checkWheelStates
                  Mode.calculateTravelThrottleThreshold(lTargetAngle.Value);

lWheelA.Target := Mode.calculateWheelTargetAngle(lWheelA,lTargetAngle.Value,SteerWheelBase,SteerWheelTrack,lInputProcessed);
lWheelB.Target := Mode.calculateWheelTargetAngle(lWheelB,lTargetAngle.Value,SteerWheelBase,SteerWheelTrack,lInputProcessed);
lWheelC.Target := Mode.calculateWheelTargetAngle(lWheelC,lTargetAngle.Value,SteerWheelBase,SteerWheelTrack,lInputProcessed);
lWheelD.Target := Mode.calculateWheelTargetAngle(lWheelD,lTargetAngle.Value,SteerWheelBase,SteerWheelTrack,lInputProcessed);

(*lWheelA.checkWheelState();
lWheelB.checkWheelState();
lWheelC.checkWheelState();
lWheelD.checkWheelState();*)

lCurrentPositiveDelta := -1000.0;
lCurrentPositiveDelta := MAX(lCurrentPositiveDelta,lWheelA.lDelta);
lCurrentPositiveDelta := MAX(lCurrentPositiveDelta,lWheelB.lDelta);
lCurrentPositiveDelta := MAX(lCurrentPositiveDelta,lWheelC.lDelta);
lCurrentPositiveDelta := MAX(lCurrentPositiveDelta,lWheelD.lDelta);

lCurrentNegativeDelta := 1000;
lCurrentNegativeDelta := MIN(lCurrentNegativeDelta,lWheelA.lDelta);
lCurrentNegativeDelta := MIN(lCurrentNegativeDelta,lWheelB.lDelta);
lCurrentNegativeDelta := MIN(lCurrentNegativeDelta,lWheelC.lDelta);
lCurrentNegativeDelta := MIN(lCurrentNegativeDelta,lWheelD.lDelta);

lCurrentAbsDelta := 0;
lCurrentAbsDelta := MAX(lCurrentAbsDelta,ABS(lWheelA.lDelta));
lCurrentAbsDelta := MAX(lCurrentAbsDelta,ABS(lWheelB.lDelta));
lCurrentAbsDelta := MAX(lCurrentAbsDelta,ABS(lWheelC.lDelta));
lCurrentAbsDelta := MAX(lCurrentAbsDelta,ABS(lWheelD.lDelta));

lStationary := (lWheelA.Stationary AND
	lWheelB.Stationary AND
	lWheelC.Stationary AND
	lWheelD.Stationary);

lStalledSubSystemsPrevious := lStalledSubSystems;
lStalledSubSystems := (lWheelA.Stalled OR
	lWheelB.Stalled OR
	lWheelC.Stalled OR
	lWheelD.Stalled);
	
lAdjustState := MAX(lWheelA.State,
	MAX(lWheelB.State,
	MAX(lWheelC.State,lWheelD.State)));
	
lModeChange := ((lWheelA.ModeChange) OR
	(lWheelB.ModeChange) OR
	(lWheelC.ModeChange) OR
	(lWheelD.ModeChange));
	
IF ((lEnableSequentialModeChange) AND (lModeChange)) THEN
	IF (NOT(lWheelD.ModeChange)) THEN
		lWheelD.ModeChangeDisableControl := FALSE;
		lWheelA.ModeChangeDisableControl := FALSE;
	END_IF
	IF (NOT(lWheelC.ModeChange)) THEN
		lWheelC.ModeChangeDisableControl := FALSE;
		lWheelD.ModeChangeDisableControl := FALSE;
	END_IF
	IF (NOT(lWheelB.ModeChange)) THEN
		lWheelB.ModeChangeDisableControl := FALSE;
		lWheelC.ModeChangeDisableControl := FALSE;
	END_IF
	IF (NOT(lWheelA.ModeChange)) THEN
		lWheelA.ModeChangeDisableControl := FALSE;
		lWheelB.ModeChangeDisableControl := FALSE;
	END_IF
ELSE
	lWheelA.ModeChangeDisableControl := FALSE;	
	lWheelB.ModeChangeDisableControl := FALSE;	
	lWheelC.ModeChangeDisableControl := FALSE;	
	lWheelD.ModeChangeDisableControl := FALSE;	
END_IF

IF (NOT(lModeChange)) THEN
	lSteerModeDiagnostic := cSteerModeDiagnosticOK;
ELSE
	IF (lEnableActiveOnModeChange) THEN
		gSystemPrimary.Active.registerActive();
	END_IF	
END_IF

                
END_METHOD

METHOD getMode : REFERENCE TO SteerMode
  VAR_INPUT
    mode : t_steer_mode;
  END_VAR
                  getMode REF= lSteerMode4WS;	

CASE mode OF		
	cSteerMode4WS:
		getMode REF= lSteerMode4WS;	
	cSteerModeLateral:
		getMode REF= lSteerModeLateral;
	cSteerModeCarousel:
		getMode REF= lSteerModeCarousel;
	cSteerModeReconfigure:
		getMode REF= lSteerModeReconfigure;
	cSteerModeLateralPos90:
		getMode REF= lSteerModeLateral;
	cSteerModeLateralNeg90:
		getMode REF= lSteerModeLateral;
	cSteerModeCustom:
		getMode REF= lSteerModeCustom;
END_CASE

                
END_METHOD

METHOD initialize
                  Name := 'Steer';

lVREnableRelativeSteering.initializeValueReference(lEnableRelativeSteering,NopSelf,'EnblRelative','Relative steering control is enabled','',cValueStyleParameter);
lVREnableZeroTargetAngleSwitch.initializeValueReference(lEnableZeroTargetAngleSwitch,NopSelf,'EnblZero','Zero target angle switch is enabled','',cValueStyleParameter);
lVREnableSequentialModeChange.initializeValueReference(lEnableSequentialModeChange,NopSelf,'EnblSeqMdChng','Sequential mode change is enabled','',cValueStyleParameter);
lVREnableActiveOnModeChange.initializeValueReference(lEnableActiveOnModeChange,NopSelf,'EnblActMdChng','Mode change has active checks enabled','',cValueStyleParameter);
lVREnableDerivedTargetAngleIncrement.initializeValueReference(lEnableDerivedTargetAngleIncrement,NopSelf,'EnblDerTrgAng','Derived target angle increment is enabled','',cValueStyleParameter);
lVREnableOperatingModeLockOnSteerModeChange.initializeValueReference(lEnableOperatingModeLockOnSteerModeChange,NopSelf,'EnblOpMdLck','Mode change has operating mode checks enabled','',cValueStyleParameter);

_Throttle.Name := 'Throttle';
lThrottle REF= _Throttle;
registerNonOperational(ADR(_Throttle));

WheelA.Name := 'mA';
WheelA.SubSystem := cSubsystemSteerA;
WheelA.ID := 1;
registerNonOperational(ADR(lWheelA));

WheelB.Name := 'mB';
WheelB.SubSystem := cSubsystemSteerB;
WheelB.ID := 2;
registerNonOperational(ADR(lWheelB));

WheelC.Name := 'mC';
WheelC.SubSystem := cSubsystemSteerC;
WheelC.ID := 3;
registerNonOperational(ADR(lWheelC));

WheelD.Name := 'mD';
WheelD.SubSystem := cSubsystemSteerD;
WheelD.ID := 4;
registerNonOperational(ADR(lWheelD));

lSteerMode4WS.Available := TRUE;
lSteerMode4WS.Enabled := TRUE;
registerNonOperational(ADR(lSteerMode4WS));

lSteerModeLateral.Available := TRUE;
lSteerModeLateral.Enabled := TRUE;
registerNonOperational(ADR(lSteerModeLateral));

lSteerModeCarousel.Available := TRUE;
lSteerModeCarousel.Enabled := TRUE;
registerNonOperational(ADR(lSteerModeCarousel));

lSteerModeReconfigure.Available := TRUE;
lSteerModeReconfigure.Enabled := FALSE;
registerNonOperational(ADR(lSteerModeReconfigure));

lSteerModeCustom.Available := TRUE;
lSteerModeCustom.Enabled := TRUE;
registerNonOperational(ADR(lSteerModeCustom));

lTargetAngle.Name := 'TargetAngle';
registerNonOperational(ADR(lTargetAngle));

lZeroTargetAngleSwitch.Name := 'ZeroTarget';
registerNonOperational(ADR(lZeroTargetAngleSwitch));

SUPER^.initialize();
SubSystem := cSubsystemSteer;

setCarouselAngle();

lEnableSequentialModeChange := FALSE;

cSteerAngleMaxUpdateDelta := 0.06; // limit on how far away the target can be pushed
cSteerAngleMaxDerivedUpdateDelta := 0.07;
cSteerAngleThrottleIncrement := 0.006;
cSteerAngleDeltaGain := 0.0;

WheelA.ControlFeedbackSign := -1.0;
WheelA.CarouselSign := 1.0;
WheelA.StandardSign := 1.0;
WheelA.DriveWheel := TRUE;
WheelA.InnerFlag := FALSE;
WheelA.WheelDirection := 1.0;
WheelA.IndependentWheels := TRUE;

WheelB.ControlFeedbackSign := -1.0;
WheelB.CarouselSign := -1.0;
WheelB.StandardSign := 1.0;
WheelB.DriveWheel := TRUE;
WheelB.InnerFlag := TRUE;
WheelB.WheelDirection := -1.0;
WheelB.IndependentWheels := TRUE;

WheelC.ControlFeedbackSign := -1.0;
WheelC.CarouselSign := 1.0;
WheelC.StandardSign := -1.0;
WheelC.DriveWheel := TRUE;
WheelC.InnerFlag := TRUE;
WheelC.WheelDirection := -1.0;
WheelC.IndependentWheels := TRUE;

WheelD.ControlFeedbackSign := -1.0;
WheelD.CarouselSign := -1.0;
WheelD.StandardSign := -1.0;
WheelD.DriveWheel := TRUE;
WheelD.InnerFlag := FALSE;
WheelD.WheelDirection := 1.0;
WheelD.IndependentWheels := TRUE;

{IF defined (TargetD19)}
	lEnableSequentialModeChange := TRUE;

	cSteerAngleMaxUpdateDelta := 0.07; // limit on how far away the target can be pushed
	cSteerAngleMaxDerivedUpdateDelta := 0.07;
	cSteerAngleThrottleIncrement := 0.08;
	cSteerAngleDeltaGain := 1.0; // foobar

	WheelA.ControlFeedbackSign := 1.0;
	WheelA.CarouselSign := 1.0;
	WheelA.StandardSign := 1.0;
	WheelA.DriveWheel := FALSE;
	WheelA.InnerFlag := FALSE;
	WheelA.WheelDirection := 1.0;
	WheelA.IndependentWheels := TRUE;

